// TIA Portal V16 export
// export: Created 2023-02-26T15:55:10.3538181Z, ExportSetting WithDefaults, DisplayName Totally Integrated Automation Portal, DisplayVersion V16 Update 3, DisplayName TIA Portal Version Control Interface, DisplayVersion V16 Update 2, DisplayName TIA Portal Openness, DisplayVersion V16 Update 3, DisplayName STEP 7 Professional, DisplayVersion V16 Update 3, DisplayName STEP 7 Safety, DisplayVersion V16, DisplayName WinCC Professional, DisplayVersion V16 Update 3
FUNCTION "FC19511_StdDebugInst1Order" : Void   // FC19511, LAD
TITLE = Standard Module [DEBUG] — First Order Response Simulation
{ S7_Optimized_Access := 'TRUE' }
AUTHOR : M_Gledhill
FAMILY : Debug
NAME : StdDebugInst1Order
VERSION : 0.1
// PRACTICAL SERIES AUTOMATION LIBRARY (PAL)   —   COPYRIGHT 2020 – M. GLEDHILL (MIT LICENCE)
//                   ———— ◆ ————
// FULL ONLINE DOCUMENTATION IS AVAILABLE AT: https://practicalseries.com/2001-pal/index.html
// stored: AutoNumber false, IsIECCheckEnabled true, SetENOAutomatically false, UDAEnableTagReadback false
   VAR_INPUT
      SYS_SIGNALS : "UT21000_Dy_SysSignals";   // Common system signals — logic and timing signals
      TRIGGER : Bool;   // Starts the simulation (rising edge starts the sim)
      INPUT : Real;   // The input function, x in the calculations
   END_VAR
   VAR_OUTPUT
      OUTPUT : Real;   // The output response, y in the calculations
   END_VAR
   VAR_IN_OUT
      DYNAMIC_DATA : "UT39511_Dy_DebugInst1Order";   // Dynamic data storage (UDT)
   END_VAR
   VAR_TEMP
      revInfo : "UT01000_St_SysRevision";   // Revision information for this block
      licInfo : "UT01001_St_SysLicence";   // Licensing information for this block
      act_CPUTime : DTL;   // Current CPU time (this block call)
      cal_01 : Real;   // Partial calculation see § 3.5 for details
      cal_02 : Real;   // Partial calculation see § 3.5 for details
      cal_03 : Real;   // Partial calculation see § 3.5 for details
      cal_04 : Real;   // Partial calculation see § 3.5 for details
      cal_05 : Real;   // Partial calculation see § 3.5 for details
      cal_06 : Real;   // Partial calculation see § 3.5 for details
      wrkElapsedTime : LTime;   // Working storage area (current elapsed time)
      wrkDeltaTime : LTime;   // Working storage area (current ΔT)
      wrkInt : Int;   // Working storage area (integer)
      wrkLInt : ULInt;   // Working storage area (long integer)
      wrkReal : Real;   // Working storage (real)
   END_VAR
   VAR CONSTANT
      k_NEG_MAX : Real := 3.4E-38;   // Largest negative number available to the REAL type
   END_VAR
   VAR_TEMP   // added for the SCL form of the ladder/FBD networks
      _w1 : Bool;
   END_VAR
BEGIN

REGION Network 1: Block description — Sections 1 to 2 inclusive
   // ▄▄▄▄▄▄▄▄▄▄▄▄▄▄▄▄▄▄▄▄▄▄▄▄▄▄▄▄▄▄▄▄▄  ＳＴＡＮＤＡＲＤ  ▄▄ 
   // 
   // 
   // TITLE:    DEBUG — FIRST ORDER RESPONSE SIMULATION
   // 
   // 
   // ▀▀▀▀▀▀▀▀▀▀▀▀▀▀▀▀▀▀▀▀▀▀▀▀▀▀▀▀▀▀▀▀▀▀▀▀▀▀▀▀▀▀▀▀ 
   // 
   // ┌──────────────────────────────────────────┐
   // │                                          │
   // │          FC19511 — SOFTWARE MODULE DESIGN SPECIFICATION (SMDS)            │
   // │                                          │
   // │      The PDF version of the SMDS for this module is available online here:        │
   // │              https://psop.uk/pal-smds-fc19511-p               │
   // │                                          │
   // │      It is also available as part of the Project User Defined Documentation,      │
   // │      it can be accessed by selecting this module in the Project Tree          │
   // │      (on the left) and pressing SHIFT+F1                        │
   // │                                          │
   // └─────────────────────────────────────── ʷᴵᴰ⁻ᶜᵇᶻ ┘
   // 
   // FC19511_StdDebugInst1Order is a debug simulation subroutine.
   // 
   // The module simulates a first order process reaction in response to an input signal.
   // 
   // The simulation is adjustable in terms of the system gain and the system time constant.
   // The output of the first order response simulation is in the form of a real number and is 
   // constrained to the resolution and range limits applicable to this number type within the Siemens 
   // Simatic S7-1500 controller.
   // 
   // The module will simulate a 1st order response to any type of input signal (step, ramp, sinusoid, 
   // freeform &c.).
   // 
   // The module also has a manual mode that can simulate an output at any specific time in 
   // response to a step input.
   // 
   // 
   // 
   // 
   // 
   // ▄▄▄▄▄▄▄▄▄▄▄▄▄▄▄▄▄▄▄▄▄▄▄▄▄▄▄▄▄▄▄▄▄▄▄▄▄▄▄▄▄▄▄▄
   // 1.     BLOCK TECHNICAL SUMMARY
   // 
   // 
   //  ――――――――――――――――――――――――――――――――――――――――――
   //  NOMENCLATURE & ADDRESSING
   //  ――――――――――――――――――――――――――――――――――――――――――
   //  BLOCK TITLE         1st Order Response Simulation
   //  BLOCK FUNCTION GROUP    Debug  
   //  BLOCK ADDRESS       FC19511
   //  BLOCK SYMBOL        FC19511_StdDebugInst1Order
   //  BLOCK USER ID         StdDebugInst1Order
   // 
   //  ――――――――――――――――――――――――――――――――――――――――――
   //  BLOCK TYPE & USAGE
   //  ――――――――――――――――――――――――――――――――――――――――――
   //  BLOCK TYPE         Function (FC)
   //  BLOCK NUMBER        19511
   //  LANGUAGE           LAD
   //  OPTIMISED ACCESS     Yes
   //  PAL USAGE TYPE       Standard block
   // 
   //  ――――――――――――――――――――――――――――――――――――――――――
   //  METRICS
   //  ――――――――――――――――――――――――――――――――――――――――――
   //  EXECUTION TIME        091.0 μs¹    (Note: = 14.4µs if TRIGGER is FALSE)
   //  LOAD MEMORY       46.0 kB
   //  WORK MEMORY           0.9 kB  
   //  ――――――――――――――――――――――――――――――――――――――――――
   //                ¹ Measured on: CPU-1515-2PN (order no. 6ES7512-2AM02-0AB0) 
   //                             https://psop.uk/pal-ds-cpu1515
   // 
   // 
   // 
   // ▂▂▂▂▂▂▂▂▂▂▂▂▂▂▂▂▂▂▂▂▂▂▂▂▂▂▂▂▂▂▂▂▂▂▂▂▂▂▂▂▂▂▂▂
   // 1.1      Additional referenced documents
   // 
   // 
   // In addition to the documents referenced in OB1 (section DOCUMENT REFERENCES), the 
   // following documents are associated with this module:
   // 
   // 
   //  ――――――――――――――――――――――――――――――――――――――――――
   //  REF.     DOCUMENT NO.         TITLE
   //  ――――――――――――――――――――――――――――――――――――――――――
   //  101  PS2001-5-2331-fc19511      FC19511 Calculation Sheet
   //  102  PS2001-5-2331-fc19511-011    FC19511 1st Order Response Simulation Spreadsheet
   //  ――――――――――――――――――――――――――――――――――――――――――
   // 
   // 
   // 
   //                ━━━   ⬙⬙⬙⬙⬙⬙   ━━━
   // 
   // 
   // 
   // ▄▄▄▄▄▄▄▄▄▄▄▄▄▄▄▄▄▄▄▄▄▄▄▄▄▄▄▄▄▄▄▄▄▄▄▄▄▄▄▄▄▄▄▄
   // 2.     FUNCTIONAL DESCRIPTION
   // 
   // 
   // ████████████████████████████████████████████
   // █                                          █
   // █ Note:   The following descriptions are taken from the associated Software Module     █
   // █     Design Specification [PS2001-5-2312-fc19511], the SMDS contains various     █
   // █     graphs that cannot be easily reproduced in these module comments. Where    █
   // █     essential, some rudimentary images have been included; however,        █
   // █     these are better viewed directly in the SMDS.                   █
   // █                                          █
   // █     Where images of the graphs are included, these are generated using           █
   // █     the Unicode braille characters and were generated by the following web site:     █
   // █     https://505e06b2.github.io/Image-to-Braille/                  █
   // █     (the images are 100 braille characters wide)                   █
   // █                                          █
   // █     The SMDS can be accessed directly by selecting this module (FC19511) in the     █
   // █     Project Tree (on the left) and pressing SHIFT+F1.                 █
   // █                                          █
   // █      The PDF version of the SMDS for this module is available online here:        █
   // █              https://psop.uk/pal-smds-fc19511-p               █
   // █                                          █
   // ████████████████████████████████████████████
   // 
   // FC19511 is the 1st Order Response Simulation module. The purpose of this module is to simulate 
   // a “first order” process reaction in response to an input signal.
   // 
   // First order systems are the most common type of system response for process control systems 
   // (for example the response generated when heating a tank of liquid). First order systems are often 
   // referred to as “first order lag” systems and generally reflect systems whereby the response of the 
   // system (the temperature of the water in the above example) follows the input (the temperature 
   // of the heating element) but with some delay (or lag). First order systems do not produce an 
   // oscillatory response to a step change of input and do not overshoot the input.
   // 
   // First order systems are so called because the equation linking the input to the out-put is always 
   // defined by a first order differential equation.
   // 
   // The following graphs show typical first order responses to a step change input:
   // 
   // 
   // 
   // Output y(t)
   // │⠄⠄⠄⠄⠄⠄⠄⠄⠄⠄⠄⠄⠄⠄⠄⠄⠄⠄⠄⠄⠄⠄⠄⠄⠄⠄⠄⠄⠄⠄⠄⠄⠄⠄⠄⠄⠄⠄⠄⠄⠄⠄⠄⠄⠄⠄⠄⠄⠄⠄⠄⠄⠄⠄⠄⠄⠄⠄⠄⠄⠄⠄⠄⠄⠄⠄⠄⠄⠄⠄⠄⠄⠄⠄⠄⠄⠄⠄⠄⠄⠄⠄⠄⠄⠄⠄⠄⠄⠄⠄⠄⠄⠄⠄⠄⠄⠄⠄⠄⠄
   // │⠤⠤⠤⠤⠤⠤⠤⠤⠤⠤⠤⠤⠤⠤⠤⠤⠤⠤⠤⠤⠤⠤⠤⠤⠤⠤⠤⠤⠤⠤⠤⠤⠤⠤⠤⠤⠤⠤⠤⠤⠤⠤⠤⠤⠤⠤⠤⠤⠤⠤⠤⢀⣀⣀⣀⣀⣀⣠⣤⣤⣤⣤⣤⣤⣤⣤⣤⣤⣤⣤⣤⣤⣤⣤⣤⠤⠤⠤⠤⠤⠤⠤⠤⠤⠤⠤⠤⠤⠤⠤⠤⠤⠤⠤⠤⠤⠤⠤⠤⠤
   // │⡇⠄⠄⠄⠄⠄⠄⠄⠄⠄⠄⠄⠄⠄⠄⠄⠄⠄⠄⠄⠄⠄⠄⠄⠄⠄⠄⠄⠄⠄⠄⠄⠄⠄⠄⠄⠄⠄⠄⣀⣀⣤⣤⡶⠶⠶⠒⠒⠛⠉⠉⠉⠉⠉⠉⠉⠉⠉⠉⠁⠄⠄⠄⠄⠄⠄⠄⠄⠄⠄⠄⠄⠄⠄⠄⠄⠄⠄⠄⠄⠄⠄⠄⠄⠄⠄⠄⠄⠄⠄⠄⠄⠄⠄⠄⠄⠄⠄⠄⠄
   // │⡇←— STEP INPUT  ⠄⠄⠄⠄⠄⠄⠄⠄⠄⠄⠄⠄⠄⠄⠄⠄⠄⠄⠄⠄⣀⣤⡶⠖⠚⠉⠉⠉⠁⠄⠄⠄⠄⠄⠄⠄⠄⠄⠄⠄⠄⠄⠄⠄⠄⠄⠄⠄⠄⠄⠄⠄⠄⠄⠄⠄⠄⠄⠄⠄⠄⠄⠄⠄⠄⠄⠄⠄⠄⠄⠄⠄⠄⠄⠄⠄⠄⠄⠄⠄⠄⠄⠄⠄⠄⠄⠄
   // │⡇⠄⠄⠄⠄⠄⠄⠄⠄⠄⠄⠄⠄⠄⠄⠄⠄⠄⠄⠄⠄⠄⠄⠄⠄⠄⠄⠄⢀⣠⡴⠖⠋⠉⠁⠄⠄⠄⠄⠄⠄⠄⠄⠄⠄⠄⠄⠄⠄⠄⠄⠄⠄⠄⠄⠄⠄⠄⠄⠄⠄⠄⠄⠄⠄⠄⠄⠄⠄⠄⠄⠄⠄⠄⠄⠄⠄⠄⠄⠄⠄⠄⠄⠄⠄⠄⠄⠄⠄⠄⠄⠄⠄⠄⠄⠄⠄⠄⠄⠄
   // │⡇⠄⠄⠄⠄⠄⠄⠄⠄⠄⠄⠄⠄⠄⠄⠄⠄⠄⠄⠄⠄⠄⠄⠄⠄⠄⣠⠾⠋⠄⠄⠄⠄⠄⠄⠄⠄⠄⠄⠄⠄⠄⠄⠄⠄⠄⠄⠄⠄⠄⠄⠄⠄⠄⠄⠄⠄⠄⠄⠄⠄⠄⠄⠄⠄⠄⠄⠄⠄⠄⠄⠄⠄⠄⠄⠄⠄⠄⠄⠄⠄⠄⠄⠄⠄⠄⠄⠄⠄⠄⠄⠄⠄⠄⠄⠄⠄⠄⠄⠄
   // │⡇⠄⠄⠄⠄⠄⠄⠄⠄⠄⠄⠄⠄⠄⠄⠄⠄⠄⠄⠄⠄⠄⠄⣀⡴⠋⠁⠄⠄⠄⠄⠄⠄⠄⠄⠄⠄⠄⠄⠄⠄⠄⠄⠄⠄⠄⠄⠄⠄⠄⠄⠄⠄⠄⠄⠄⠄⠄⠄⠄⠄⠄⠄⠄⠄⠄⠄⠄⠄⠄⠄⠄⠄⠄⠄⠄⠄⠄⠄⠄⠄⠄⠄⠄⠄⠄⠄⠄⠄⠄⠄⠄⠄⠄⠄⠄⠄⠄⠄⠄
   // │⡇⠄⠄⠄⠄⠄⠄⠄⠄⠄⠄⠄⠄⠄⠄⠄⠄⠄⠄⠄⠄⣠⠾⠁←— DELAYED OUTPUT  ⠄⠄⠄⠄⠄⠄⠄⠄⠄⠄⠄⠄⠄⠄⠄⠄⠄⠄⠄⠄⠄⠄⠄⠄⠄⠄⠄⠄⠄⠄⠄⠄⠄⠄⠄⠄⠄⠄⠄⠄⠄⠄⠄⠄⠄⠄⠄⠄⠄⠄⠄⠄⠄⠄⠄⠄⠄⠄
   // │⡇⠄⠄⠄⠄⠄⠄⠄⠄⠄⠄⠄⠄⠄⠄⠄⠄⠄⠄⢀⡴⠏⠄⠄⠄⠄⠄⠄⠄⠄⠄⠄⠄⠄⠄⠄⠄⠄⠄⠄⠄⠄⠄⠄⠄⠄⠄⠄⠄⠄⠄⠄⠄⠄⠄⠄⠄⠄⠄⠄⠄⠄⠄⠄⠄⠄⠄⠄⠄⠄⠄⠄⠄⠄⠄⠄⠄⠄⠄⠄⠄⠄⠄⠄⠄⠄⠄⠄⠄⠄⠄⠄⠄⠄⠄⠄⠄⠄⠄⠄
   // │⡇⠄⠄⠄⠄⠄⠄⠄⠄⠄⠄⠄⠄⠄⠄⠄⠄⢀⣴⠏⠄⠄⠄⠄⠄⠄⠄⠄⠄⠄⠄⠄⠄⠄⠄⠄⠄⠄⠄⠄⠄⠄⠄⠄⠄⠄⠄⠄⠄⠄⠄⠄⠄⠄⠄⠄⠄⠄⠄⠄⠄⠄⠄⠄⠄⠄⠄⠄⠄⠄⠄⠄⠄⠄⠄⠄⠄⠄⠄⠄⠄⠄⠄⠄⠄⠄⠄⠄⠄⠄⠄⠄⠄⠄⠄⠄⠄⠄⠄⠄
   // │⡇⠄⠄⠄⠄⠄⠄⠄⠄⠄⠄⠄⠄⠄⠄⠄⢠⡜⠃⠄⠄⠄⠄⠄⠄⠄⠄⠄⠄⠄⠄⠄⠄⠄⠄⠄⠄⠄⠄⠄⠄⠄⠄⠄⠄⠄⠄⠄⠄⠄⠄⠄⠄⠄⠄⠄⠄⠄⠄⠄⠄⠄⠄⠄⠄⠄⠄⠄⠄⠄⠄⠄⠄⠄⠄⠄⠄⠄⠄⠄⠄⠄⠄⠄⠄⠄⠄⠄⠄⠄⠄⠄⠄⠄⠄⠄⠄⠄⠄⠄
   // │⡇⠄⠄⠄⠄⠄⠄⠄⠄⠄⠄⠄⠄⠄⠄⢰⠟⠁⠄⠄⠄⠄⠄⠄⠄⠄⠄⠄⠄⠄⠄⠄⠄⠄⠄⠄⠄⠄⠄⠄⠄⠄⠄⠄⠄⠄⠄⠄⠄⠄⠄⠄⠄⠄⠄⠄⠄⠄⠄⠄⠄⠄⠄⠄⠄⠄⠄⠄⠄⠄⠄⠄⠄⠄⠄⠄⠄⠄⠄⠄⠄⠄⠄⠄⠄⠄⠄⠄⠄⠄⠄⠄⠄⠄⠄⠄⠄⠄⠄⠄
   // │⡇⠄⠄⠄⠄⠄⠄⠄⠄⠄⠄⠄⠄⠄⣰⡏⠄⠄⠄⠄⠄⠄⠄⠄⠄⠄⠄⠄⠄⠄⠄⠄⠄⠄⠄⠄⠄⠄⠄⠄⠄⠄⠄⠄⠄⠄⠄⠄⠄⠄⠄⠄⠄⠄⠄⠄⠄⠄⠄⠄⠄⠄⠄⠄⠄⠄⠄⠄⠄⠄⠄⠄⠄⠄⠄⠄⠄⠄⠄⠄⠄⠄⠄⠄⠄⠄⠄⠄⠄⠄⠄⠄⠄⠄⠄⠄⠄⠄⠄⠄
   // │⡇⠄⠄⠄⠄⠄⠄⠄⠄⠄⠄⠄⠄⢠⠏⠄⠄⠄⠄⠄⠄⠄⠄⠄⠄⠄⠄⠄⠄⠄⠄⠄⠄⠄⠄⠄⠄⠄⠄⠄⠄⠄⠄⠄⠄⠄⠄⠄⠄⠄⠄⠄⠄⠄⠄⠄⠄⠄⠄⠄⠄⠄⠄⠄⠄⠄⠄⠄⠄⠄⠄⠄⠄⠄⠄⠄⠄⠄⠄⠄⠄⠄⠄⠄⠄⠄⠄⠄⠄⠄⠄⠄⠄⠄⠄⠄⠄⠄⠄⠄
   // │⡇⠄⠄⠄⠄⠄⠄⠄⠄⠄⠄⠄⣰⡟⠄⠄⠄⠄⠄⠄⠄⠄⠄⠄⠄⠄⠄⠄⠄⠄⠄⠄⠄⠄⠄⠄⠄⠄⠄⠄⠄⠄⠄⠄⠄⠄⠄⠄⠄⠄⠄⠄⠄⠄⠄⠄⠄⠄⠄⠄⠄⠄⠄⠄⠄⠄⠄⠄⠄⠄⠄⠄⠄⠄⠄⠄⠄⠄⠄⠄⠄⠄⠄⠄⠄⠄⠄⠄⠄⠄⠄⠄⠄⠄⠄⠄⠄⠄⠄⠄
   // │⡇⠄⠄⠄⠄⠄⠄⠄⠄⠄⠄⢠⠏⠄⠄⠄⠄⠄⠄⠄⠄⠄⠄⠄⠄⠄⠄⠄⠄⠄⠄⠄⠄⠄⠄⠄⠄⠄⠄⠄⠄⠄⠄⠄⠄⠄⠄⠄⠄⠄⠄⠄⠄⠄⠄⠄⠄⠄⠄⠄⠄⠄⠄⠄⠄⠄⠄⠄⠄⠄⠄⠄⠄⠄⠄⠄⠄⠄⠄⠄⠄⠄⠄⠄⠄⠄⠄⠄⠄⠄⠄⠄⠄⠄⠄⠄⠄⠄⠄⠄
   // │⡇⠄⠄⠄⠄⠄⠄⠄⠄⠄⢠⡿⠄⠄⠄⠄⠄⠄⠄⠄⠄⠄⠄⠄⠄⠄⠄⠄⠄⠄⠄⠄⠄⠄⠄⠄⠄⠄⠄⠄⠄⠄⠄⠄⠄⠄⠄⠄⠄⠄⠄⠄⠄⠄⠄⠄⠄⠄⠄⠄⠄⠄⠄⠄⠄⠄⠄⠄⠄⠄⠄⠄⠄⠄⠄⠄⠄⠄⠄⠄⠄⠄⠄⠄⠄⠄⠄⠄⠄⠄⠄⠄⠄⠄⠄⠄⠄⠄⠄⠄
   // │⡇⠄⠄⠄⠄⠄⠄⠄⠄⠄⡿⠁⠄⠄⠄⠄⠄⠄⠄⠄⠄⠄⠄⠄⠄⠄⠄⠄⠄⠄⠄⠄⠄⠄⠄⠄⠄⠄⠄⠄⠄⠄⠄⠄⠄⠄⠄⠄⠄⠄⠄⠄⠄⠄⠄⠄⠄⠄⠄⠄⠄⠄⠄⠄⠄⠄⠄⠄⠄⠄⠄⠄⠄⠄⠄⠄⠄⠄⠄⠄⠄⠄⠄⠄⠄⠄⠄⠄⠄⠄⠄⠄⠄⠄⠄⠄⠄⠄⠄⠄
   // │⡇⠄⠄⠄⠄⠄⠄⠄⠄⣼⠃⠄⠄⠄⠄⠄⠄⠄⠄⠄⠄⠄⠄⠄⠄⠄⠄⠄⠄⠄⠄⠄⠄⠄⠄⠄⠄⠄⠄⠄⠄⠄⠄⠄⠄⠄⠄⠄⠄⠄⠄⠄⠄⠄⠄⠄⠄⠄⠄⠄⠄⠄⠄⠄⠄⠄⠄⠄⠄⠄⠄⠄⠄⠄⠄⠄⠄⠄⠄⠄⠄⠄⠄⠄⠄⠄⠄⠄⠄⠄⠄⠄⠄⠄⠄⠄⠄⠄⠄⠄
   // │⡇⠄⠄⠄⠄⠄⠄⠄⢰⡟⠄⠄⠄⠄⠄⠄⠄⠄⠄⠄⠄⠄⠄⠄⠄⠄⠄⠄⠄⠄⠄⠄⠄⠄⠄⠄⠄⠄⠄⠄⠄⠄⠄⠄⠄⠄⠄⠄⠄⠄⠄⠄⠄⠄⠄⠄⠄⠄⠄⠄⠄⠄⠄⠄⠄⠄⠄⠄⠄⠄⠄⠄⠄⠄⠄⠄⠄⠄⠄⠄⠄⠄⠄⠄⠄⠄⠄⠄⠄⠄⠄⠄⠄⠄⠄⠄⠄⠄⠄⠄
   // │⡇⠄⠄⠄⠄⠄⠄⠄⡞⠄⠄⠄⠄⠄⠄⠄⠄⠄⠄⠄⠄⠄⠄⠄⠄⠄⠄⠄⠄⠄⠄⠄⠄⠄⠄⠄⠄⠄⠄⠄⠄⠄⠄⠄⠄⠄⠄⠄⠄⠄⠄⠄⠄⠄⠄⠄⠄⠄⠄⠄⠄⠄⠄⠄⠄⠄⠄⠄⠄⠄⠄⠄⠄⠄⠄⠄⠄⠄⠄⠄⠄⠄⠄⠄⠄⠄⠄⠄⠄⠄⠄⠄⠄⠄⠄⠄⠄⠄⠄⠄
   // │⡇⠄⠄⠄⠄⠄⠄⣰⡇⠄⠄⠄⠄⠄⠄⠄⠄⠄⠄⠄⠄⠄⠄⠄⠄⠄⠄⠄⠄⠄⠄⠄⠄⠄⠄⠄⠄⠄⠄⠄⠄⠄⠄⠄⠄⠄⠄⠄⠄⠄⠄⠄⠄⠄⠄⠄⠄⠄⠄⠄⠄⠄⠄⠄⠄⠄⠄⠄⠄⠄⠄⠄⠄⠄⠄⠄⠄⠄⠄⠄⠄⠄⠄⠄⠄⠄⠄⠄⠄⠄⠄⠄⠄⠄⠄⠄⠄⠄⠄⠄
   // │⡇⠄⠄⠄⠄⠄⢰⡟⠄⠄⠄⠄⠄⠄⠄⠄⠄⠄⠄⠄⠄⠄⠄⠄⠄⠄⠄⠄⠄⠄⠄⠄⠄⠄⠄⠄⠄⠄⠄⠄⠄⠄⠄⠄⠄⠄⠄⠄⠄⠄⠄⠄⠄⠄⠄⠄⠄⠄⠄⠄⠄⠄⠄⠄⠄⠄⠄⠄⠄⠄⠄⠄⠄⠄⠄⠄⠄⠄⠄⠄⠄⠄⠄⠄⠄⠄⠄⠄⠄⠄⠄⠄⠄⠄⠄⠄⠄⠄⠄⠄
   // │⡇⠄⠄⠄⠄⠄⣸⠁⠄⠄⠄⠄⠄⠄⠄⠄⠄⠄⠄⠄⠄⠄⠄⠄⠄⠄⠄⠄⠄⠄⠄⠄⠄⠄⠄⠄⠄⠄⠄⠄⠄⠄⠄⠄⠄⠄⠄⠄⠄⠄⠄⠄⠄⠄⠄⠄⠄⠄⠄⠄⠄⠄⠄⠄⠄⠄⠄⠄⠄⠄⠄⠄⠄⠄⠄⠄⠄⠄⠄⠄⠄⠄⠄⠄⠄⠄⠄⠄⠄⠄⠄⠄⠄⠄⠄⠄⠄⠄⠄⠄
   // │⡇⠄⠄⠄⠄⢠⡇⠄⠄⠄⠄⠄⠄⠄⠄⠄⠄⠄⠄⠄⠄⠄⠄⠄⠄⠄⠄⠄⠄⠄⠄⠄⠄⠄⠄⠄⠄⠄⠄⠄⠄⠄⠄⠄⠄⠄⠄⠄⠄⠄⠄⠄⠄⠄⠄⠄⠄⠄⠄⠄⠄⠄⠄⠄⠄⠄⠄⠄⠄⠄⠄⠄⠄⠄⠄⠄⠄⠄⠄⠄⠄⠄⠄⠄⠄⠄⠄⠄⠄⠄⠄⠄⠄⠄⠄⠄⠄⠄⠄⠄
   // │⡇⠄⠄⠄⠄⣿⠃⠄⠄⠄⠄⠄⠄⠄⠄⠄⠄⠄⠄⠄⠄⠄⠄⠄⠄⠄⠄⠄⠄⠄⠄⠄⠄⠄⠄⠄⠄⠄⠄⠄⠄⠄⠄⠄⠄⠄⠄⠄⠄⠄⠄⠄⠄⠄⠄⠄⠄⠄⠄⠄⠄⠄⠄⠄⠄⠄⠄⠄⠄⠄⠄⠄⠄⠄⠄⠄⠄⠄⠄⠄⠄⠄⠄⠄⠄⠄⠄⠄⠄⠄⠄⠄⠄⠄⠄⠄⠄⠄⠄⠄
   // │⡇⠄⠄⠄⢸⡏⠄⠄⠄⠄⠄⠄⠄⠄⠄⠄⠄⠄⠄⠄⠄⠄⠄⠄⠄⠄⠄⠄⠄⠄⠄⠄⠄⠄⠄⠄⠄⠄⠄⠄⠄⠄⠄⠄⠄⠄⠄⠄⠄⠄⠄⠄⠄⠄⠄⠄⠄⠄⠄⠄⠄⠄⠄⠄⠄⠄⠄⠄⠄⠄⠄⠄⠄⠄⠄⠄⠄⠄⠄⠄⠄⠄⠄⠄⠄⠄⠄⠄⠄⠄⠄⠄⠄⠄⠄⠄⠄⠄⠄⠄
   // │⡇⠄⠄⠄⣸⠁⠄⠄⠄⠄⠄⠄⠄⠄⠄⠄⠄⠄⠄⠄⠄⠄⠄⠄⠄⠄⠄⠄⠄⠄⠄⠄⠄⠄⠄⠄⠄⠄⠄⠄⠄⠄⠄⠄⠄⠄⠄⠄⠄⠄⠄⠄⠄⠄⠄⠄⠄⠄⠄⠄⠄⠄⠄⠄⠄⠄⠄⠄⠄⠄⠄⠄⠄⠄⠄⠄⠄⠄⠄⠄⠄⠄⠄⠄⠄⠄⠄⠄⠄⠄⠄⠄⠄⠄⠄⠄⠄⠄⠄⠄
   // │⡇⠄⠄⢠⡇⠄⠄⠄⠄⠄⠄⠄⠄⠄⠄⠄⠄⠄⠄⠄⠄⠄⠄⠄⠄⠄⠄⠄⠄⠄⠄⠄⠄⠄⠄⠄⠄⠄⠄⠄⠄⠄⠄⠄⠄⠄⠄⠄⠄⠄⠄⠄⠄⠄⠄⠄⠄⠄⠄⠄⠄⠄⠄⠄⠄⠄⠄⠄⠄⠄⠄⠄⠄⠄⠄⠄⠄⠄⠄⠄⠄⠄⠄⠄⠄⠄⠄⠄⠄⠄⠄⠄⠄⠄⠄⠄⠄⠄⠄⠄
   // │⡇⠄⠄⣼⠇⠄⠄⠄⠄⠄⠄⠄⠄⠄⠄⠄⠄⠄⠄⠄⠄⠄⠄⠄⠄⠄⠄⠄⠄⠄⠄⠄⠄⠄⠄⠄⠄⠄⠄⠄⠄⠄⠄⠄⠄⠄⠄⠄⠄⠄⠄⠄⠄⠄⠄⠄⠄⠄⠄⠄⠄⠄⠄⠄⠄⠄⠄⠄⠄⠄⠄⠄⠄⠄⠄⠄⠄⠄⠄⠄⠄⠄⠄⠄⠄⠄⠄⠄⠄⠄⠄⠄⠄⠄⠄⠄⠄⠄⠄⠄
   // │⡇⠄⠄⡿⠄⠄⠄⠄⠄⠄⠄⠄⠄⠄⠄⠄⠄⠄⠄⠄⠄⠄⠄⠄⠄⠄⠄⠄⠄⠄⠄⠄⠄⠄⠄⠄⠄⠄⠄⠄⠄⠄⠄⠄⠄⠄⠄⠄⠄⠄⠄⠄⠄⠄⠄⠄⠄⠄⠄⠄⠄⠄⠄⠄⠄⠄⠄⠄⠄⠄⠄⠄⠄⠄⠄⠄⠄⠄⠄⠄⠄⠄⠄⠄⠄⠄⠄⠄⠄⠄⠄⠄⠄⠄⠄⠄⠄⠄⠄⠄
   // │⡇⠄⢰⠃⠄⠄⠄⠄⠄⠄⠄⠄⠄⠄⠄⠄⠄⠄⠄⠄⠄⠄⠄⠄⠄⠄⠄⠄⠄⠄⠄⠄⠄⠄⠄⠄⠄⠄⠄⠄⠄⠄⠄⠄⠄⠄⠄⠄⠄⠄⠄⠄⠄⠄⠄⠄⠄⠄⠄⠄⠄⠄⠄⠄⠄⠄⠄⠄⠄⠄⠄⠄⠄⠄⠄⠄⠄⠄⠄⠄⠄⠄⠄⠄⠄⠄⠄⠄⠄⠄⠄⠄⠄⠄⠄⠄⠄⠄⠄⠄
   // │⡇⠄⣾⠄⠄⠄⠄⠄⠄⠄⠄⠄⠄⠄⠄⠄⠄⠄⠄⠄⠄⠄⠄⠄⠄⠄⠄⠄⠄⠄⠄⠄⠄⠄⠄⠄⠄⠄⠄⠄⠄⠄⠄⠄⠄⠄⠄⠄⠄⠄⠄⠄⠄⠄⠄⠄⠄⠄⠄⠄⠄⠄⠄⠄⠄⠄⠄⠄⠄⠄⠄⠄⠄⠄⠄⠄⠄⠄⠄⠄⠄⠄⠄⠄⠄⠄⠄⠄⠄⠄⠄⠄⠄⠄⠄⠄⠄⠄⠄⠄
   // │⡇⢰⡟⠄⠄⠄⠄⠄⠄⠄⠄⠄⠄⠄⠄⠄⠄⠄⠄⠄⠄⠄⠄⠄⠄⠄⠄⠄⠄⠄⠄⠄⠄⠄⠄⠄⠄⠄⠄⠄⠄⠄⠄⠄⠄⠄⠄⠄⠄⠄⠄⠄⠄⠄⠄⠄⠄⠄⠄⠄⠄⠄⠄⠄⠄⠄⠄⠄⠄⠄⠄⠄⠄⠄⠄⠄⠄⠄⠄⠄⠄⠄⠄⠄⠄⠄⠄⠄⠄⠄⠄⠄⠄⠄⠄⠄⠄⠄⠄⠄
   // │⡇⣾⠇⠄⠄⠄⠄⠄⠄⠄⠄⠄⠄⠄⠄⠄⠄⠄⠄⠄⠄⠄⠄⠄⠄⠄⠄⠄⠄⠄⠄⠄⠄⠄⠄⠄⠄⠄⠄⠄⠄⠄⠄⠄⠄⠄⠄⠄⠄⠄⠄⠄⠄⠄⠄⠄⠄⠄⠄⠄⠄⠄⠄⠄⠄⠄⠄⠄⠄⠄⠄⠄⠄⠄⠄⠄⠄⠄⠄⠄⠄⠄⠄⠄⠄⠄⠄⠄⠄⠄⠄⠄⠄⠄⠄⠄⠄⠄⠄⠄
   // │⡇⡿⠄⠄⠄⠄⠄⠄⠄⠄⠄⠄⠄⠄⠄⠄⠄⠄⠄⠄⠄⠄⠄⠄⠄⠄⠄⠄⠄⠄⠄⠄⠄⠄⠄⠄⠄⠄⠄⠄⠄⠄⠄⠄⠄⠄⠄⠄⠄⠄⠄⠄⠄⠄⠄⠄⠄⠄⠄⠄⠄⠄⠄⠄⠄⠄⠄⠄⠄⠄⠄⠄⠄⠄⠄⠄⠄⠄⠄⠄⠄⠄⠄⠄⠄⠄⠄⠄⠄⠄⠄⠄⠄⠄⠄⠄⠄⠄⠄⠄
   // │⡇⠃⠄⠄⠄⠄⠄⠄⠄⠄⠄⠄⠄⠄⠄⠄⠄⠄⠄⠄⠄⠄⠄⠄⠄⠄⠄⠄⠄⠄⠄⠄⠄⠄⠄⠄⠄⠄⠄⠄⠄⠄⠄⠄⠄⠄⠄⠄⠄⠄⠄⠄⠄⠄⠄⠄⠄⠄⠄⠄⠄⠄⠄⠄⠄⠄⠄⠄⠄⠄⠄⠄⠄⠄⠄⠄⠄⠄⠄⠄⠄⠄⠄⠄⠄⠄⠄⠄⠄⠄⠄⠄⠄⠄⠄⠄⠄⠄⠄⠄
   // ┼ ─ ─ ─ ─ ─ ─ ─ ─ ─ ─ ─ ─ ─ ─ ─ ─ ─ ─ ─ ─ ─ ─ ─ ─ ─ ─ ─ ─ ─ ─ ─ ─ ─ ─ ─ ─ ─ ─ ─ ─ ─ ─  ─ ─ ─ ─    Time (t)
   // 
   // 
   // 
   // ▂▂▂▂▂▂▂▂▂▂▂▂▂▂▂▂▂▂▂▂▂▂▂▂▂▂▂▂▂▂▂▂▂▂▂▂▂▂▂▂▂▂▂▂
   // 2.1      Scope and limitations of the simulation
   // 
   // 
   // The first order response simulation will provide a real time response for a first order simulation.
   // 
   // The simulation will be adjustable in terms of the system gain (K) and the time constant of the 
   // system (τ).
   // 
   // The output of the first order response simulation will be in the form of a real number.
   // 
   // 
   // 
   // 
   // ▁▁▁▁▁▁▁▁▁▁▁▁▁▁▁▁▁▁▁▁▁▁▁▁▁▁▁▁▁▁▁▁▁▁▁▁▁▁▁▁▁▁▁▁
   // 2.1.1     The limitations of the simulation
   // 
   // 
   // The output of the second order response simulation will be in the form of a real number and will 
   // be constrained to the limits applicable to this number type within the Siemens controller.
   // 
   // The S7-1500 range of Controllers supports real numbers as values, these are 32-bit numbers 
   // and, within a Controller, have the following range limits:
   // 
   // 
   //  ――――――――――――――――――――――――――――――――――――――――――
   //              LOWER RANGE LIMIT     UPPER RANGE LIMIT
   //  ――――――――――――――――――――――――――――――――――――――――――
   //  S7-1500 real number:     ±3.402323×10^(-38)           ±3.402323×10^(+38)
   //  ――――――――――――――――――――――――――――――――――――――――――
   // 
   // This range is considered acceptable for all practical uses of the module.
   // 
   // 
   // 
   // ▁▁▁▁▁▁▁▁▁▁▁▁▁▁▁▁▁▁▁▁▁▁▁▁▁▁▁▁▁▁▁▁▁▁▁▁▁▁▁▁▁▁▁▁
   // 2.1.2     The nature of the simulation calculations
   // 
   // 
   // The module will generate the correct responses for any first order system. The module uses a 
   // discrete time approximation calculation to determine the correct output for any given input. The 
   // calculation is an iterative algorithm, the formulae for which is derived in full in the associated 
   // calculations sheet [Ref. 101], available here:
   // 
   //          https://psop.uk/pal-calc-fc19511-p
   // 
   // These calculations are based around the mathematical functions available to the Controller 
   // (these are in addition to the standard mathematical operations: addition, subtraction, 
   // multiplication and division).
   // 
   // Each Controller supports the following common mathematical functions:
   // 
   // 
   //  ――――――――――――――――――――――――――――――――――――――――――
   //  OPERATION    EXAMPLE         DESCRIPTION
   //  ――――――――――――――――――――――――――――――――――――――――――
   //  SQR        x^2          Form the square
   //  SQRT         √x            Form the square root
   //  EXP        e^x          Exponential
   //  LN          log_e(⁡x)        Natural logarithm
   //  SIN         sin(⁡x)         Sine
   //  ASIN          sin^-1(x)          Arcsine, inverse sine
   //  COS          cos(⁡x)        Cosine
   //  ACOS        cos^-1(x)         Arccosine, inverse cosine
   //  TAN           tan(⁡x)         Tangent
   //  ATAN         tan^-1(x)         Arctangent, inverse tangent
   //  ABS        |x|            Modulus
   //  ――――――――――――――――――――――――――――――――――――――――――
   //  Table 2.1 S7 Controller — common mathematical functions
   // 
   // 
   // 
   // ▂▂▂▂▂▂▂▂▂▂▂▂▂▂▂▂▂▂▂▂▂▂▂▂▂▂▂▂▂▂▂▂▂▂▂▂▂▂▂▂▂▂▂▂
   // 2.2      The second order response
   // 
   // 
   // The response of a second order system (y) to an input (x) is defined using the general form of a 
   // second order system transfer function, this is expressed below in the time domain as a second 
   // order differential equation (see the calculation sheet [Ref. 101], Appendix B for details):
   // 
   //                 dy
   //             τ ----- ┼  y  =  Kx  (2.1)
   //                 dt
   // 
   // Where:    K is the system gain
   //      τ is referred to as the system time constant (seconds)
   // 
   // 
   // 
   // ▂▂▂▂▂▂▂▂▂▂▂▂▂▂▂▂▂▂▂▂▂▂▂▂▂▂▂▂▂▂▂▂▂▂▂▂▂▂▂▂▂▂▂▂
   // 2.3      The calculations
   // 
   // 
   // Two forms of calculation are needed to produce a model for a first order system. The first being a 
   // continuous simulation running in real-time with a varying or constant input signal.
   // 
   // The second being the discrete result for a step input under manual conditions (i.e. a fixed input 
   // and specific time are provided and a single, corresponding output value generated).
   // 
   // Both of these calculations are discussed in the following sections:
   // 
   // 
   // 
   // ▁▁▁▁▁▁▁▁▁▁▁▁▁▁▁▁▁▁▁▁▁▁▁▁▁▁▁▁▁▁▁▁▁▁▁▁▁▁▁▁▁▁▁▁
   // 2.3.1     Real-time simulation calculation for any input type
   // 
   // 
   // The normal operation of the module (in automatic mode) is to produce a continuous real-time 
   // model of a first order system that once triggered, runs continuously, producing an output 
   // response that mimics a first order system responding to a variable (or constant) input as time 
   // progresses, the simulation continues until the triggering condition is removed.
   // 
   // The calculation needed to produce a first order system response to any type of input signal is 
   // best achieved using a discrete time approximation method. The details of this method are given 
   // in [Ref. 101], Section 2.1, and the results are given below:
   // 
   // The final form of the calculations that will be used in the FC19511 software module for a real time 
   // simulation to any input type is:
   // 
   //    y[n] = Ka x[n]  ┼ (1-a) y[n-1]  (2.2)
   // 
   //              ΔT
   //    where:   a = ----------
   //            τ+ΔT
   // 
   //    K is the system gain (a constant number)
   //    τ is the system time constant (in seconds)
   //    Δt is the sampling interval between calculations (in seconds)
   //    x[n] is the input at the current iteration 
   //    y[n] is the output at the current iteration 
   //    y[n-1] is the output at the previous iteration 
   // 
   // 
   // It should be noted that this is an iterative algorithm, the previous value of the output must 
   // be retained between calculations.
   // 
   // For best results, Δt should be very much smaller than the system time constant, i.e.:
   // 
   //                    τ
   //    Δt ≪ τ      Typically, Δt ≤ ----
   //                      10
   // 
   // Note also, that Δt need not be constant between samples.
   // 
   // 
   // 
   // ▁▁▁▁▁▁▁▁▁▁▁▁▁▁▁▁▁▁▁▁▁▁▁▁▁▁▁▁▁▁▁▁▁▁▁▁▁▁▁▁▁▁▁▁
   // 2.3.2     Manual simulation calculation for a step input at a particular time
   // 
   // 
   // In manual mode, an instantaneous calculation is carried out using the first order equation at a 
   // particular time and for a particular input value.
   // 
   // Since, under manual control, both the time and the input are fixed single values, it is not possible 
   // to determine the nature of the input (i.e. is it a ramp, sinusoid &c.), hence for all manual 
   // operations within the simulation, the input is considered to be a step input that changed to the 
   // manually specified input value at time = 0, and that prior to this the input was zero¹. I.e. a step 
   // input that changed from zero to the specified value at time = 0.
   // 
   // To produce a specific output value in response to a fixed step input at a particular time, it is 
   // necessary to solve the first order differential equation given in equation (2.1), as a non-iterative, 
   // discreate calculation. To do this, it is necessary to convert the equation into the Laplace domain² 
   // (using standard Laplace transforms, see [Ref. 101], Appendix A) algebraically solve the equation 
   // and then convert the result back to the time domain (using the standard inverse Laplace 
   // transforms, again see [Ref. 101], Appendix A).
   // 
   // The final form of the manual calculations that will be used in the FC19511 software module for a 
   // single point input type is:
   // 
   //          ┌      -t/τ  ┐
   //    y(t) = KX│ 1 ─  e   │
   //          └       ┘
   // 
   //    K is the system gain (a constant number)
   //    τ is the system time constant (in seconds)
   //    X is the fixed input value
   // 
   // 
   // ――――――――――
   // ¹         A step response is the most common type of response
   // 
   // ²         The calculation sheet associated with this module [Ref. 101], explains the Laplace 
   //      transform mechanisms and how they are used within the calculations necessary for 
   //      the functioning of this module. Further explanation of the Laplace transform is not 
   //      given in this document, again the reader is referred to the calculation 
   //      sheet [Ref. 101].
   // ――――――――――
   // 
   // 
   // 
   // ▁▁▁▁▁▁▁▁▁▁▁▁▁▁▁▁▁▁▁▁▁▁▁▁▁▁▁▁▁▁▁▁▁▁▁▁▁▁▁▁▁▁▁▁
   // 2.3.3     Calculation spreadsheet model
   // 
   // 
   // An accompanying spreadsheet [Ref. 016] is available, this allows all the various responses to be 
   // graphically simulated with adjustable values (it was this spreadsheet that produced the various 
   // response plots used within this document), this spreadsheet is available here:
   // 
   //      http://psop.uk/pal-calc-fc19511-p
   // 
   // 
   // 
   // ▂▂▂▂▂▂▂▂▂▂▂▂▂▂▂▂▂▂▂▂▂▂▂▂▂▂▂▂▂▂▂▂▂▂▂▂▂▂▂▂▂▂▂▂
   // 2.4      Real-time responses for typical inputs
   // 
   // 
   // First order systems respond to various types of input (step, ramp, sinusoidal) in very predictable 
   // ways. First order systems never produce oscillatory responses (unless the input itself is 
   // oscillating) and never overshoot the input (cf. 2nd order systems, see FC19512). The general 
   // response of a first order system is that of an inherent delay (or lag) in the response of the output 
   // compared with the input.
   // 
   // This inherent delay is reflected in the system time constant (τ), measured in seconds.
   // 
   // The following sections consider how the system time constant affects the output for several 
   // typical input types:
   // 
   // 
   // STEP INPUT
   // 
   // │⠄⠄⠄⠄⠄⠄⠄⠄⠄⠄⠄⠄⠄⠄⠄⠄⠄⠄⠄⠄⠄⠄⠄τ = 20s⠄⠄⠄⠄⠄⠄⠄⠄⠄⠄⠄⠄⠄⠄⠄⠄⠄⠄⠄⠄⠄⠄⠄⠄⠄⠄⠄⠄⠄⠄⠄⠄⠄⠄⠄⠄⠄⠄⠄⠄⠄⠄⠄⠄⠄⠄⠄⠄⠄⠄⠄⠄⠄⠄⠄⠄⠄⠄⠄⠄⠄⠄⠄⠄⠄⠄⠄⠄⠄⠄⠄⠄
   // X─ ─ ─ ─ ─ ─ ─ ─ ─ ─ ─ ─ ─ ─ ─ ─ ─ ─ ─ ─ ─ ─ ─ ─ ─ ─ ─ ─ ─ ─ ─ ─ ─ ─ ─ ─ ─ ─ ─ ─ ─ ─ ─ ─ ─ ─ ─
   // │⠄⠄⠄⠄⠄⠄⠄⠄⠄⠄⠄⠄⠄⠄⠄⠄⠄⠄⠄⠄⠄⠄⠄⠄⠄⠄⠄⠄⠄⠄⠄⠄⠄⠄⠄⠄⠄⠄⠄⠄⠄⠄⠄⠄⠄⠄⠄⠄⠄⠄⠄⠄⠄⠄⠄⠄⠄⠄⠄⠄⠄⣀⣀⣀⣀⣠⣤⡤⠤⠤⠶⠶⠶⠶⠒⠒⠒⠒⠚⠛⠛⠛⠛⠉⠉⠉⠉⠉⠉⠉⠉⠉⠉⠉⠉⠉⠉⠉⠉⠉
   // │⠄⠄⠄⠄⠄⠄⠄⠄⠄⠄⠄⠄⠄⠄⠄⠄⠄⠄⠄⠄⠄⠄⠄⠄⠄⠄⠄⠄⠄⠄⠄⠄⠄⠄⠄⠄⠄⠄⠄⠄⠄⠄⠄⠄⠄⠄⠄⠄⠄⠄⢀⣀⣠⡤⠤⠶⠖⠒⠛⠄⠄⠄⠄⠄⠄⠄⠄⠄⠄⠄⠄⠄⠄⠄99% of steady state ─ ─ ─ ─ ╎⠄
   // │⠄⠄⠄⠄⠄⠄⠄⠄⠄⠄⠄⠄⠄⠄⠄⠄⠄⠄⠄⠄⠄⠄⠄⠄⠄⠄⠄⠄⠄⠄⠄⠄⠄⠄⠄⠄⠄⠄⠄⠄⠄⠄⠄⢀⣀⣠⠴⠖⠚⠋⠉⠁⠄⠄⠄⠄⠄⠄⠄⠄⠄⠄⠄⠄⠄⠄⠄⠄⠄⠄⠄⠄⠄⠄⠄⠄⠄⠄⠄⠄⠄⠄⠄⠄⠄⠄⠄⠄⠄⠄⠄⠄⠄⠄⠄⠄⠄⠄╎⠄
   // │⠄⠄⠄⠄⠄⠄⠄⠄⠄⠄⠄⠄⠄⠄⠄⠄⠄⠄⠄⠄⠄⠄⠄⠄⠄⠄⠄⠄⠄⠄⠄⠄⠄⠄⠄⠄⠄⠄⢀⣠⡤⠖⠚⠉⠁⠄⠄⠄⠄⠄⠄⠄⠄⠄⠄⠄⠄⠄⠄⠄⠄⠄⠄⠄⠄⠄⠄⠄⠄⠄⠄⠄⠄⠄⠄⠄⠄⠄⠄⠄⠄⠄⠄⠄⠄⠄⠄⠄⠄⠄⠄⠄⠄⠄⠄⠄⠄⠄╎⠄
   // │⠄⠄⠄⠄⠄⠄⠄⠄⠄⠄⠄⠄⠄⠄⠄⠄⠄⠄⠄⠄⠄⠄⠄⠄⠄⠄⠄⠄⠄⠄⠄⠄⠄⠄⠄⣠⡴⠚⠋⠁⠄⠄⠄⠄⠄⠄⠄⠄⠄⠄⠄⠄⠄⠄⠄⠄⠄⠄⠄⠄⠄⠄⠄⠄⠄⠄⠄⠄⠄⠄⠄⠄⠄⠄⠄⠄⠄⠄⠄⠄⠄⠄⠄⠄⠄⠄⠄⠄⠄⠄⠄⠄⠄⠄⠄⠄⠄⠄╎⠄
   // │⠄⠄⠄⠄⠄⠄⠄⠄⠄⠄⠄⠄⠄⠄⠄⠄⠄⠄⠄⠄⠄⠄⠄⠄⠄⠄⠄⠄⠄⠄⠄⢀⣠⠖⠋⠁⠄⠄⠄⠄⠄⠄⠄⠄⠄⠄⠄⠄⠄⠄⠄⠄⠄⠄⠄⠄⠄⠄⠄⠄⠄⠄⠄⠄⠄⠄⠄⠄⠄⠄⠄⠄⠄⠄⠄⠄⠄⠄⠄⠄⠄⠄⠄⠄⠄⠄⠄⠄⠄⠄⠄⠄⠄⠄⠄⠄⠄⠄╎⠄
   // │⠄⠄⠄⠄⠄⠄⠄⠄⠄⠄⠄⠄⠄⠄⠄⠄⠄⠄⠄⠄⠄⠄⠄⠄⠄⠄⠄⠄⠄⣠⠴⠋⠄⠄⠄⠄⠄⠄⠄⠄⠄⠄⠄⠄⠄⠄⠄⠄⠄⠄⠄⠄⠄⠄⠄⠄⠄⠄⠄⠄⠄⠄⠄⠄⠄⠄⠄⠄⠄⠄⠄⠄⠄⠄⠄⠄⠄⠄⠄⠄⠄⠄⠄⠄⠄⠄⠄⠄⠄⠄⠄⠄⠄⠄⠄⠄⠄⠄╎⠄
   // │⠄⠄⠄⠄⠄⠄⠄⠄⠄⠄⠄⠄⠄⠄⠄⠄⠄⠄⠄⠄⠄⠄⠄⠄⠄⠄⢀⡤⠚⠁⠄⠄⠄⠄⠄⠄⠄⠄⠄⠄⠄⠄⠄⠄⠄⠄⠄⠄⠄⠄⠄⠄⠄⠄⠄⠄⠄⠄⠄⠄⠄⠄⠄⠄⠄⠄⠄⠄⠄⠄⠄⠄⠄⠄⠄⠄⠄⠄⠄⠄⠄⠄⠄⠄⠄⠄⠄⠄⠄⠄⠄⠄⠄⠄⠄⠄⠄⠄╎⠄
   // │⠄⠄⠄⠄⠄⠄⠄⠄⠄⠄⠄⠄⠄⠄⠄⠄⠄⠄⠄⠄⠄⠄⠄⠄⢀⡴⠋⠄⠄⠄⠄⠄⠄⠄⠄⠄⠄⠄⠄⠄⠄⠄⠄⠄⠄⠄⠄⠄⠄⠄⠄⠄⠄⠄⠄⠄⠄⠄⠄⠄⠄⠄⠄⠄⠄⠄⠄⠄⠄⠄⠄⠄⠄⠄⠄⠄⠄⠄⠄⠄⠄⠄⠄⠄⠄⠄⠄⠄⠄⠄⠄⠄⠄⠄⠄⠄⠄⠄╎⠄
   // │⠄⠄⠄⠄⠄⠄⠄⠄⠄⠄⠄⠄⠄⠄⠄⠄⠄⠄⠄⠄⠄⠄⢀⡴⠋⠄⠄⠄⠄⠄⠄⠄⠄⠄⠄⠄⠄⠄⠄⠄⠄⠄⠄⠄⠄⠄⠄⠄⠄⠄⠄⠄⠄⠄⠄⠄⠄⠄⠄⠄⠄⠄⠄⠄⠄⠄⠄⠄⠄⠄⠄⠄⠄⠄⠄⠄⠄⠄⠄⠄⠄⠄⠄⠄⠄⠄⠄⠄⠄⠄⠄⠄⠄⠄⠄⠄⠄⠄╎⠄
   // │⠄⠄⠄⠄⠄⠄⠄⠄⠄⠄⠄⠄⠄⠄⠄⠄⠄⠄⠄⠄⠄⣠⠋⠄⠄⠄⠄⠄⠄⠄⠄⠄⠄⠄⠄⠄⠄⠄⠄⠄⠄⠄⠄⠄⠄⠄⠄⠄⠄⠄⠄⠄⠄⠄⠄⠄⠄⠄⠄⠄⠄⠄⠄⠄⠄⠄⠄⠄⠄⠄⠄⠄⠄⠄⠄⠄⠄⠄⠄⠄⠄⠄⠄⠄⠄⠄⠄⠄⠄⠄⠄⠄⠄⠄⠄⠄⠄⠄╎⠄
   // │⠄⠄⠄⠄⠄⠄⠄⠄⠄⠄⠄⠄⠄⠄⠄⠄⠄⠄⠄⢀⠞⠁⠄⠄⠄⠄⠄⠄⠄⠄⠄⠄⠄⠄⠄⠄⠄⠄⠄⠄⠄⠄⠄⠄⠄⠄⠄⠄⠄⠄⠄⠄⠄⠄⠄⠄⠄⠄⠄⠄⠄⠄⠄⠄⠄⠄⠄⠄⠄⠄⠄⠄⠄⠄⠄⠄⠄⠄⠄⠄⠄⠄⠄⠄⠄⠄⠄⠄⠄⠄⠄⠄⠄⠄⠄⠄⠄⠄╎⠄
   // │⠄⠄⠄⠄⠄⠄⠄⠄⠄⠄⠄⠄⠄⠄⠄⠄⠄⠄⣴⠋─ ─ ─ ─ ─  63% of steady state  ⠄⠄⠄⠄⠄⠄⠄⠄⠄⠄⠄⠄⠄⠄⠄⠄⠄⠄⠄⠄⠄⠄⠄⠄⠄⠄⠄⠄⠄⠄⠄⠄⠄⠄⠄⠄⠄⠄⠄⠄⠄⠄⠄⠄⠄⠄⠄⠄⠄⠄⠄╎⠄
   // │⠄⠄⠄⠄⠄⠄⠄⠄⠄⠄⠄⠄⠄⠄⠄⠄⢀⡾⠁⠄⠄⠄⠄⠄⠄⠄⠄⠄⠄⠄⠄⠄⠄⠄⠄⠄⠄⠄⠄⠄⠄⠄⠄⠄⠄⠄⠄⠄⠄⠄⠄⠄⠄⠄⠄⠄⠄⠄⠄⠄⠄⠄⠄⠄⠄⠄⠄⠄⠄⠄⠄⠄⠄⠄⠄⠄⠄⠄⠄⠄⠄⠄⠄⠄⠄⠄⠄⠄⠄⠄⠄⠄⠄⠄⠄⠄⠄⠄╎⠄
   // │⠄⠄⠄⠄⠄⠄⠄⠄⠄⠄⠄⠄⠄⠄⠄⢠⠞⠄ ╎⠄⠄⠄⠄⠄⠄⠄⠄⠄⠄⠄⠄⠄⠄⠄⠄⠄⠄⠄⠄⠄⠄⠄⠄⠄⠄⠄⠄⠄⠄⠄⠄⠄⠄⠄⠄⠄⠄⠄⠄⠄⠄⠄⠄⠄⠄⠄⠄⠄⠄⠄⠄⠄⠄⠄⠄⠄⠄⠄⠄⠄⠄⠄⠄⠄⠄⠄⠄⠄⠄⠄⠄⠄⠄⠄⠄⠄⠄╎⠄
   // │⠄⠄⠄⠄⠄⠄⠄⠄⠄⠄⠄⠄⠄⠄⣠⠏⠄⠄ ╎⠄⠄⠄⠄⠄⠄⠄⠄⠄⠄⠄⠄⠄⠄⠄⠄⠄⠄⠄⠄⠄⠄⠄⠄⠄⠄⠄⠄⠄⠄⠄⠄⠄⠄⠄⠄⠄⠄⠄⠄⠄⠄⠄⠄⠄⠄⠄⠄⠄⠄⠄⠄⠄⠄⠄⠄⠄⠄⠄⠄⠄⠄⠄⠄⠄⠄⠄⠄⠄⠄⠄⠄⠄⠄⠄⠄⠄⠄╎⠄
   // │⠄⠄⠄⠄⠄⠄⠄⠄⠄⠄⠄⠄⠄⣰⠋⠄⠄⠄ ╎⠄⠄⠄⠄⠄⠄⠄⠄⠄⠄⠄⠄⠄⠄⠄⠄⠄⠄⠄⠄⠄⠄⠄⠄⠄⠄⠄⠄⠄⠄⠄⠄⠄⠄⠄⠄⠄⠄⠄⠄⠄⠄⠄⠄⠄⠄⠄⠄⠄⠄⠄⠄⠄⠄⠄⠄⠄⠄⠄⠄⠄⠄⠄⠄⠄⠄⠄⠄⠄⠄⠄⠄⠄⠄⠄⠄⠄⠄╎⠄
   // │⠄⠄⠄⠄⠄⠄⠄⠄⠄⠄⠄⠄⣰⠃⠄⠄⠄⠄ ╎⠄⠄⠄⠄⠄⠄⠄⠄⠄⠄⠄⠄⠄⠄⠄⠄⠄⠄⠄⠄⠄⠄⠄⠄⠄⠄⠄⠄⠄⠄⠄⠄⠄⠄⠄⠄⠄⠄⠄⠄⠄⠄⠄⠄⠄⠄⠄⠄⠄⠄⠄⠄⠄⠄⠄⠄⠄⠄⠄⠄⠄⠄⠄⠄⠄⠄⠄⠄⠄⠄⠄⠄⠄⠄⠄⠄⠄⠄╎⠄
   // │⠄⠄⠄⠄⠄⠄⠄⠄⠄⠄⠄⣸⠃⠄⠄⠄⠄⠄ ╎⠄⠄⠄⠄⠄⠄⠄⠄⠄⠄⠄⠄⠄⠄⠄⠄⠄⠄⠄⠄⠄⠄⠄⠄⠄⠄⠄⠄⠄⠄⠄⠄⠄⠄⠄⠄⠄⠄⠄⠄⠄⠄⠄⠄⠄⠄⠄⠄⠄⠄⠄⠄⠄⠄⠄⠄⠄⠄⠄⠄⠄⠄⠄⠄⠄⠄⠄⠄⠄⠄⠄⠄⠄⠄⠄⠄⠄⠄╎⠄
   // │⠄⠄⠄⠄⠄⠄⠄⠄⠄⠄⣰⠃⠄⠄⠄⠄⠄⠄ ╎⠄⠄⠄⠄⠄⠄⠄⠄⠄⠄⠄⠄⠄⠄⠄⠄⠄⠄⠄⠄⠄⠄⠄⠄⠄⠄⠄⠄⠄⠄⠄⠄⠄⠄⠄⠄⠄⠄⠄⠄⠄⠄⠄⠄⠄⠄⠄⠄⠄⠄⠄⠄⠄⠄⠄⠄⠄⠄⠄⠄⠄⠄⠄⠄⠄⠄⠄⠄⠄⠄⠄⠄⠄⠄⠄⠄⠄⠄╎⠄
   // │⠄⠄⠄⠄⠄⠄⠄⠄⠄⣰⠃⠄⠄⠄⠄⠄⠄⠄ ╎⠄⠄⠄⠄⠄⠄⠄⠄⠄⠄⠄⠄⠄⠄⠄⠄⠄⠄⠄⠄⠄⠄⠄⠄⠄⠄⠄⠄⠄⠄⠄⠄⠄⠄⠄⠄⠄⠄⠄⠄⠄⠄⠄⠄⠄⠄⠄⠄⠄⠄⠄⠄⠄⠄⠄⠄⠄⠄⠄⠄⠄⠄⠄⠄⠄⠄⠄⠄⠄⠄⠄⠄⠄⠄⠄⠄⠄⠄╎⠄
   // │⠄⠄⠄⠄⠄⠄⠄⠄⢰⠇⠄⠄⠄⠄⠄⠄⠄⠄ ╎⠄⠄⠄⠄⠄⠄⠄⠄⠄⠄⠄⠄⠄⠄⠄⠄⠄⠄⠄⠄⠄⠄⠄⠄⠄⠄⠄⠄⠄⠄⠄⠄⠄⠄⠄⠄⠄⠄⠄⠄⠄⠄⠄⠄⠄⠄⠄⠄⠄⠄⠄⠄⠄⠄⠄⠄⠄⠄⠄⠄⠄⠄⠄⠄⠄⠄⠄⠄⠄⠄⠄⠄⠄⠄⠄⠄⠄⠄╎⠄
   // │⠄⠄⠄⠄⠄⠄⠄⢠⡏⠄⠄⠄⠄⠄⠄⠄⠄⠄ ╎⠄⠄⠄⠄⠄⠄⠄⠄⠄⠄⠄⠄⠄⠄⠄⠄⠄⠄⠄⠄⠄⠄⠄⠄⠄⠄⠄⠄⠄⠄⠄⠄⠄⠄⠄⠄⠄⠄⠄⠄⠄⠄⠄⠄⠄⠄⠄⠄⠄⠄⠄⠄⠄⠄⠄⠄⠄⠄⠄⠄⠄⠄⠄⠄⠄⠄⠄⠄⠄⠄⠄⠄⠄⠄⠄⠄⠄⠄╎⠄
   // │⠄⠄⠄⠄⠄⠄⠄⡞⠄⠄⠄⠄⠄⠄⠄⠄⠄⠄ ╎⠄⠄⠄⠄⠄⠄⠄⠄⠄⠄⠄⠄⠄⠄⠄⠄⠄⠄⠄⠄⠄⠄⠄⠄⠄⠄⠄⠄⠄⠄⠄⠄⠄⠄⠄⠄⠄⠄⠄⠄⠄⠄⠄⠄⠄⠄⠄⠄⠄⠄⠄⠄⠄⠄⠄⠄⠄⠄⠄⠄⠄⠄⠄⠄⠄⠄⠄⠄⠄⠄⠄⠄⠄⠄⠄⠄⠄⠄╎⠄
   // │⠄⠄⠄⠄⠄⠄⣸⠃⠄⠄⠄⠄⠄⠄⠄⠄⠄⠄ ╎⠄⠄⠄⠄⠄⠄⠄⠄⠄⠄⠄⠄⠄⠄⠄⠄⠄⠄⠄⠄⠄⠄⠄⠄⠄⠄⠄⠄⠄⠄⠄⠄⠄⠄⠄⠄⠄⠄⠄⠄⠄⠄⠄⠄⠄⠄⠄⠄⠄⠄⠄⠄⠄⠄⠄⠄⠄⠄⠄⠄⠄⠄⠄⠄⠄⠄⠄⠄⠄⠄⠄⠄⠄⠄⠄⠄⠄⠄╎⠄
   // │⠄⠄⠄⠄⠄⢰⠇⠄⠄⠄⠄⠄⠄⠄⠄⠄⠄⠄ ╎⠄⠄⠄⠄⠄⠄⠄⠄⠄⠄⠄⠄⠄⠄⠄⠄⠄⠄⠄⠄⠄⠄⠄⠄⠄⠄⠄⠄⠄⠄⠄⠄⠄⠄⠄⠄⠄⠄⠄⠄⠄⠄⠄⠄⠄⠄⠄⠄⠄⠄⠄⠄⠄⠄⠄⠄⠄⠄⠄⠄⠄⠄⠄⠄⠄⠄⠄⠄⠄⠄⠄⠄⠄⠄⠄⠄⠄⠄╎⠄
   // │⠄⠄⠄⠄⢀⡟⠄⠄⠄⠄⠄⠄⠄⠄⠄⠄⠄⠄ ╎⠄⠄⠄⠄⠄⠄⠄⠄⠄⠄⠄⠄⠄⠄⠄⠄⠄⠄⠄⠄⠄⠄⠄⠄⠄⠄⠄⠄⠄⠄⠄⠄⠄⠄⠄⠄⠄⠄⠄⠄⠄⠄⠄⠄⠄⠄⠄⠄⠄⠄⠄⠄⠄⠄⠄⠄⠄⠄⠄⠄⠄⠄⠄⠄⠄⠄⠄⠄⠄⠄⠄⠄⠄⠄⠄⠄⠄⠄╎⠄
   // │⠄⠄⠄⠄⡼⠁⠄⠄⠄⠄⠄⠄⠄⠄⠄⠄⠄⠄ ╎⠄⠄⠄⠄⠄⠄⠄⠄⠄⠄⠄⠄⠄⠄⠄⠄⠄⠄⠄⠄⠄⠄⠄⠄⠄⠄⠄⠄⠄⠄⠄⠄⠄⠄⠄⠄⠄⠄⠄⠄⠄⠄⠄⠄⠄⠄⠄⠄⠄⠄⠄⠄⠄⠄⠄⠄⠄⠄⠄⠄⠄⠄⠄⠄⠄⠄⠄⠄⠄⠄⠄⠄⠄⠄⠄⠄⠄⠄╎⠄
   // │⠄⠄⠄⢰⠇⠄⠄⠄⠄⠄⠄⠄⠄⠄⠄⠄⠄⠄ ╎⠄⠄⠄⠄⠄⠄⠄⠄⠄⠄⠄⠄⠄⠄⠄⠄⠄⠄⠄⠄⠄⠄⠄⠄⠄⠄⠄⠄⠄⠄⠄⠄⠄⠄⠄⠄⠄⠄⠄⠄⠄⠄⠄⠄⠄⠄⠄⠄⠄⠄⠄⠄⠄⠄⠄⠄⠄⠄⠄⠄⠄⠄⠄⠄⠄⠄⠄⠄⠄⠄⠄⠄⠄⠄⠄⠄⠄⠄╎⠄
   // │⠄⠄⢀⡏⠄⠄⠄⠄⠄⠄⠄⠄⠄⠄⠄⠄⠄⠄ ╎⠄⠄⠄⠄⠄⠄⠄⠄⠄⠄⠄⠄⠄⠄⠄⠄⠄⠄⠄⠄⠄⠄⠄⠄⠄⠄⠄⠄⠄⠄⠄⠄⠄⠄⠄⠄⠄⠄⠄⠄⠄⠄⠄⠄⠄⠄⠄⠄⠄⠄⠄⠄⠄⠄⠄⠄⠄⠄⠄⠄⠄⠄⠄⠄⠄⠄⠄⠄⠄⠄⠄⠄⠄⠄⠄⠄⠄⠄╎⠄
   // │⠄⠄⡼⠁⠄⠄⠄⠄⠄⠄⠄⠄⠄⠄⠄⠄⠄⠄ ╎⠄⠄⠄⠄⠄⠄⠄⠄⠄⠄⠄⠄⠄⠄⠄⠄⠄⠄⠄⠄⠄⠄⠄⠄⠄⠄⠄⠄⠄⠄⠄⠄⠄⠄⠄⠄⠄⠄⠄⠄⠄⠄⠄⠄⠄⠄⠄⠄⠄⠄⠄⠄⠄⠄⠄⠄⠄⠄⠄⠄⠄⠄⠄⠄⠄⠄⠄⠄⠄⠄⠄⠄⠄⠄⠄⠄⠄⠄╎⠄
   // │⠄⣸⠃⠄⠄⠄⠄⠄⠄⠄⠄⠄⠄⠄⠄⠄⠄⠄ ╎⠄⠄⠄⠄⠄⠄⠄⠄⠄⠄⠄⠄⠄⠄⠄⠄⠄⠄⠄⠄⠄⠄⠄⠄⠄⠄⠄⠄⠄⠄⠄⠄⠄⠄⠄⠄⠄⠄⠄⠄⠄⠄⠄⠄⠄⠄⠄⠄⠄⠄⠄⠄⠄⠄⠄⠄⠄⠄⠄⠄⠄⠄⠄⠄⠄⠄⠄⠄⠄⠄⠄⠄⠄⠄⠄⠄⠄⠄╎⠄
   // │⡴⠃⠄⠄⠄⠄⠄⠄⠄⠄⠄⠄⠄⠄⠄⠄⠄⠄ ╎⠄⠄⠄⠄⠄⠄⠄⠄⠄⠄⠄⠄⠄⠄⠄⠄⠄⠄⠄⠄⠄⠄⠄⠄⠄⠄⠄⠄⠄⠄⠄⠄⠄⠄⠄⠄⠄⠄⠄⠄⠄⠄⠄⠄⠄⠄⠄⠄⠄⠄⠄⠄⠄⠄⠄⠄⠄⠄⠄⠄⠄⠄⠄⠄⠄⠄⠄⠄⠄⠄⠄⠄⠄⠄⠄⠄⠄⠄╎⠄
   // ┼ ─ ─ ─ ─ ┼ ─ ─ ─ ─ ┼ ─ ─ ─ ─ ┼ ─ ─ ─ ─ ┼ ─ ─ ─ ─ ┼ ─ ─ ─ ─ ┼ ─ ─ ─ ─ ┼ ─ ─ ─ ─ ┼ ─ ─ ─ ─ ┼ ─ ─ ─ ─ ┼
   // 0.0     10       20       30       40       50       60       70       80       90      100 s
   //               τ                                               5τ
   //    Increasing τ gives a slower response.
   // 
   //                1
   //    Initial rate of change = ---   Time to reach 63% of input (X) = τ   Time to reach steady state = 5τ
   //                τ
   // 
   // 
   // RAMP INPUT
   // 
   // │⠄⠄⠄⠄⠄⠄⠄⠄⠄⠄⠄⠄⠄⠄⠄⠄⠄⠄⠄⠄⠄⠄⠄τ = 20s ⠄⠄⠄⠄⠄⠄⠄⠄⠄⠄⠄⠄⠄⠄⠄⠄⠄⠄⠄⠄⠄⠄⠄⠄⠄⠄⠄⠄⠄⠄⠄⠄⠄⠄⠄⠄⠄⠄⠄⠄⠄⠄⠄⠄⠄⠄⠄⠄⠄⠄⠄⠄⠄⠄⠄⠄⠄⠄⠄⠄⠄⠄⠄⠄⠄⠄⠄⠄⢀⡠⠔
   // │⠄⠄⠄⠄⠄⠄⠄⠄⠄⠄⠄⠄⠄⠄⠄⠄⠄⠄⠄⠄⠄⠄⠄⠄⠄⠄⠄⠄⠄⠄⠄⠄⠄⠄⠄⠄⠄⠄⠄⠄⠄⠄⠄⠄⠄⠄⠄⠄⠄⠄⠄⠄⠄⠄⠄⠄⠄⠄⠄⠄⠄⠄⠄⠄⠄⠄⠄⠄⠄⠄⠄⠄⠄⠄⠄⠄⠄⠄⠄⠄⠄⠄⠄⠄⠄⠄⠄⠄⠄⠄⠄⠄⠄⢀⣠⠴⠊⠉⠄⠄
   // │⠄⠄⠄⠄⠄⠄⠄⠄⠄⠄⠄⠄⠄⠄⠄⠄⠄⠄⠄⠄⠄⠄⠄⠄⠄⠄⠄⠄⠄⠄⠄⠄⠄⠄⠄⠄⠄⠄⠄⠄⠄⠄⠄⠄⠄⠄⠄⠄⠄⠄⠄⠄⠄⠄⠄⠄⠄⠄⠄⠄⠄⠄⠄⠄⠄⠄⠄⠄⠄⠄⠄⠄⠄⠄⠄⠄⠄⠄⠄⠄⠄⠄⠄⠄⠄⠄⠄⠄⠄⢀⣀⠴⠊⠉⠄⠄⠄⠄⠄⠄
   // │⠄⠄⠄⠄⠄⠄⠄⠄⠄⠄⠄⠄⠄⠄⠄⠄⠄⠄⠄⠄⠄⠄⠄⠄⠄⠄⠄⠄⠄⠄⠄⠄⠄⠄⠄⠄⠄⠄⠄⠄⠄⠄⠄⠄⠄⠄⠄⠄⠄⠄⠄⠄⠄⠄⠄⠄⠄⠄⠄⠄⠄⠄⠄⠄⠄⠄⠄⠄⠄⠄⠄⠄⠄⠄⠄⠄⠄⠄⠄⠄⠄⠄⠄⠄⠄⠄⣀⡤⠒⠋← ─ INPUT
   // │⠄⠄⠄⠄⠄⠄⠄⠄⠄⠄⠄⠄⠄⠄⠄⠄⠄⠄⠄⠄⠄⠄⠄⠄⠄⠄⠄⠄⠄⠄⠄⠄⠄⠄⠄⠄⠄⠄⠄⠄⠄⠄⠄⠄⠄⠄⠄⠄⠄⠄⠄⠄⠄⠄⠄⠄⠄⠄⠄⠄⠄⠄⠄⠄⠄⠄⠄⠄⠄⠄⠄⠄⠄⠄⠄⠄⠄⠄⠄⠄⠄⠄⢀⡤⠖⠋⠁⠄⠄⠄⠄⠄⠄⠄⠄⠄⠄⠄⠄⠄
   // │⠄⠄⠄⠄⠄⠄⠄⠄⠄⠄⠄⠄⠄⠄⠄⠄⠄⠄⠄⠄⠄⠄⠄⠄⠄⠄⠄⠄⠄⠄⠄⠄⠄⠄⠄⠄⠄⠄⠄⠄⠄⠄⠄⠄⠄⠄⠄⠄⠄⠄⠄⠄⠄⠄⠄⠄⠄⠄⠄⠄⠄⠄⠄⠄⠄⠄⠄⠄⠄⠄⠄⠄⠄⠄⠄⠄⠄⠄⢀⣠⠔⠊⠁⠄⠄⠄⠄⠄⠄⠄⠄⠄⠄⠄⠄⠄⠄⣀⣤⡾
   // │⠄⠄⠄⠄⠄⠄⠄⠄⠄⠄⠄⠄⠄⠄⠄⠄⠄⠄⠄⠄⠄⠄⠄⠄⠄⠄⠄⠄⠄⠄⠄⠄⠄⠄⠄⠄⠄⠄⠄⠄⠄⠄⠄⠄⠄⠄⠄⠄⠄⠄⠄⠄⠄⠄⠄⠄⠄⠄⠄⠄⠄⠄⠄⠄⠄⠄⠄⠄⠄⠄⠄⠄⠄⠄⢀⣠⠔⠚⠁← ─ ─  τ  ─ ─→⢀⣤⡶⠟⠋⠄⠄
   // │⠄⠄⠄⠄⠄⠄⠄⠄⠄⠄⠄⠄⠄⠄⠄⠄⠄⠄⠄⠄⠄⠄⠄⠄⠄⠄⠄⠄⠄⠄⠄⠄⠄⠄⠄⠄⠄⠄⠄⠄⠄⠄⠄⠄⠄⠄⠄⠄⠄⠄⠄⠄⠄⠄⠄⠄⠄⠄⠄⠄⠄⠄⠄⠄⠄⠄⠄⠄⠄⠄⠄⣠⠤⠚⠉⠄⠄⠄⠄⠄⠄⠄⠄⠄⠄⠄⠄⠄⠄⢀⣤⡶⠟⠋⠁⠄⠄⠄⠄⠄
   // │⠄⠄⠄⠄⠄⠄⠄⠄⠄⠄⠄⠄⠄⠄⠄⠄⠄⠄⠄⠄⠄⠄⠄⠄⠄⠄⠄⠄⠄⠄⠄⠄⠄⠄⠄⠄⠄⠄⠄⠄⠄⠄⠄⠄⠄⠄⠄⠄⠄⠄⠄⠄⠄⠄⠄⠄⠄⠄⠄⠄⠄⠄⠄⠄⠄⠄⠄⣀⡤⠒⠉⠄⠄⠄⠄⠄⠄⠄⠄⠄⠄⠄⠄⠄⠄⢀⣠⣴⠞⠋⠁⠄⠄⠄⠄⠄⠄⠄⠄⠄
   // │⠄⠄⠄⠄⠄⠄⠄⠄⠄⠄⠄⠄⠄⠄⠄⠄⠄⠄⠄⠄⠄⠄⠄⠄⠄⠄⠄⠄⠄⠄⠄⠄⠄⠄⠄⠄⠄⠄⠄⠄⠄⠄⠄⠄⠄⠄⠄⠄⠄⠄⠄⠄⠄⠄⠄⠄⠄⠄⠄⠄⠄⠄⠄⣀⡤⠖⠋⠄⠄⠄⠄⠄⠄⠄⠄⠄⠄⠄⠄⠄⠄⢀⣠⣴⠞⠛⠁← ─ OUTPUT
   // │⠄⠄⠄⠄⠄⠄⠄⠄⠄⠄⠄⠄⠄⠄⠄⠄⠄⠄⠄⠄⠄⠄⠄⠄⠄⠄⠄⠄⠄⠄⠄⠄⠄⠄⠄⠄⠄⠄⠄⠄⠄⠄⠄⠄⠄⠄⠄⠄⠄⠄⠄⠄⠄⠄⠄⠄⠄⠄⠄⣀⡠⠴⠊⠁⠄⠄⠄⠄⠄⠄⠄⠄⠄⠄⠄⠄⠄⢀⣀⣤⠶⠛⠉⠄⠄⠄⠄⠄⠄⠄⠄⠄⠄⠄⠄⠄⠄⠄⠄⠄
   // │⠄⠄⠄⠄⠄⠄⠄⠄⠄⠄⠄⠄⠄⠄⠄⠄⠄⠄⠄⠄⠄⠄⠄⠄⠄⠄⠄⠄⠄⠄⠄⠄⠄⠄⠄⠄⠄⠄⠄⠄⠄⠄⠄⠄⠄⠄⠄⠄⠄⠄⠄⠄⠄⠄⠄⢀⣀⠴⠊⠁⠄⠄⠄⠄⠄⠄⠄⠄⠄⠄⠄⠄⠄⠄⣀⣴⠶⠛⠉⠄⠄⠄⠄⠄⠄⠄⠄⠄⠄⠄⠄⠄⠄⠄⠄⠄⠄⠄⠄⠄
   // │⠄⠄⠄⠄⠄⠄⠄⠄⠄⠄⠄⠄⠄⠄⠄⠄⠄⠄⠄⠄⠄⠄⠄⠄⠄⠄⠄⠄⠄⠄⠄⠄⠄⠄⠄⠄⠄⠄⠄⠄⠄⠄⠄⠄⠄⠄⠄⠄⠄⠄⠄⠄⣀⠴⠚⠉⠄⠄⠄⠄⠄⠄⠄⠄⠄⠄⠄⠄⠄⠄⣀⣴⠶⠛⠉⠄⠄⠄⠄⠄⠄⠄⠄⠄⠄⠄⠄⠄⠄⠄⠄⠄⠄⠄⠄⠄⠄⠄⠄⠄
   // │⠄⠄⠄⠄⠄⠄⠄⠄⠄⠄⠄⠄⠄⠄⠄⠄⠄⠄⠄⠄⠄⠄⠄⠄⠄⠄⠄⠄⠄⠄⠄⠄⠄⠄⠄⠄⠄⠄⠄⠄⠄⠄⠄⠄⠄⠄⠄⠄⣀⡤⠒⠉⠁⠄⠄⠄⠄⠄⠄⠄⠄⠄⠄⠄⠄⠄⣀⣤⠶⠟⠉⠁⠄⠄⠄⠄⠄⠄⠄⠄⠄⠄⠄⠄⠄⠄⠄⠄⠄⠄⠄⠄⠄⠄⠄⠄⠄⠄⠄⠄
   // │⠄⠄⠄⠄⠄⠄⠄⠄⠄⠄⠄⠄⠄⠄⠄⠄⠄⠄⠄⠄⠄⠄⠄⠄⠄⠄⠄⠄⠄⠄⠄⠄⠄⠄⠄⠄⠄⠄⠄⠄⠄⠄⠄⠄⣀⡤⠖⠋⠁⠄⠄⠄⠄⠄⠄⠄⠄⠄⠄⠄⠄⠄⣀⣤⡶⠟⠉⠁⠄⠄⠄⠄⠄⠄⠄⠄⠄⠄⠄⠄⠄⠄⠄⠄⠄⠄⠄⠄⠄⠄⠄⠄⠄⠄⠄⠄⠄⠄⠄⠄
   // │⠄⠄⠄⠄⠄⠄⠄⠄⠄⠄⠄⠄⠄⠄⠄⠄⠄⠄⠄⠄⠄⠄⠄⠄⠄⠄⠄⠄⠄⠄⠄⠄⠄⠄⠄⠄⠄⠄⠄⠄⢀⡠⠖⠋⠁⠄⠄⠄⠄⠄⠄⠄⠄⠄⠄⠄⠄⠄⣀⣤⡶⠞⠋⠁⠄⠄⠄⠄⠄⠄⠄⠄⠄⠄⠄⠄⠄⠄⠄⠄⠄⠄⠄⠄⠄⠄⠄⠄⠄⠄⠄⠄⠄⠄⠄⠄⠄⠄⠄⠄
   // │⠄⠄⠄⠄⠄⠄⠄⠄⠄⠄⠄⠄⠄⠄⠄⠄⠄⠄⠄⠄⠄⠄⠄⠄⠄⠄⠄⠄⠄⠄⠄⠄⠄⠄⠄⠄⠄⣠⠖⠊⠉⠄⠄⠄⠄⠄⠄⠄⠄⠄⠄⠄⠄⠄⣀⣤⡶⠟⠉⠁⠄⠄⠄⠄⠄⠄⠄⠄⠄⠄⠄⠄⠄⠄⠄⠄⠄⠄⠄⠄⠄⠄⠄⠄⠄⠄⠄⠄⠄⠄⠄⠄⠄⠄⠄⠄⠄⠄⠄⠄
   // │⠄⠄⠄⠄⠄⠄⠄⠄⠄⠄⠄⠄⠄⠄⠄⠄⠄⠄⠄⠄⠄⠄⠄⠄⠄⠄⠄⠄⠄⠄⠄⠄⠄⣠⠤⠚⠉⠄⠄⠄⠄⠄⠄⠄⠄⠄⠄⠄⠄⠄⢀⣤⡶⠟⠋⠁⠄⠄⠄⠄⠄⠄⠄⠄⠄⠄⠄⠄⠄⠄⠄⠄⠄⠄⠄⠄⠄⠄⠄⠄⠄⠄⠄⠄⠄⠄⠄⠄⠄⠄⠄⠄⠄⠄⠄⠄⠄⠄⠄⠄
   // │⠄⠄⠄⠄⠄⠄⠄⠄⠄⠄⠄⠄⠄⠄⠄⠄⠄⠄⠄⠄⠄⠄⠄⠄⠄⠄⠄⠄⠄⣀⡤⠖⠋⠄⠄⠄⠄⠄⠄⠄⠄⠄⠄⠄⠄⠄⣀⣤⡶⠟⠋⠁⠄⠄⠄⠄⠄⠄⠄⠄⠄⠄⠄⠄⠄⠄⠄⠄⠄⠄⠄⠄⠄⠄⠄⠄⠄⠄⠄⠄⠄⠄⠄⠄⠄⠄⠄⠄⠄⠄⠄⠄⠄⠄⠄⠄⠄⠄⠄⠄
   // │⠄⠄⠄⠄⠄⠄⠄⠄⠄⠄⠄⠄⠄⠄⠄⠄⠄⠄⠄⠄⠄⠄⠄⠄⠄⣀⡤⠖⠋⠄⠄⠄⠄⠄⠄⠄⠄⠄⠄⠄⠄⢀⣠⣤⠾⠛⠉⠄⠄⠄⠄⠄⠄⠄⠄⠄⠄⠄⠄⠄⠄⠄⠄⠄⠄⠄⠄⠄⠄⠄⠄⠄⠄⠄⠄⠄⠄⠄⠄⠄⠄⠄⠄⠄⠄⠄⠄⠄⠄⠄⠄⠄⠄⠄⠄⠄⠄⠄⠄⠄
   // │⠄⠄⠄⠄⠄⠄⠄⠄⠄⠄⠄⠄⠄⠄⠄⠄⠄⠄⠄⠄⠄⢀⣠⠔⠋⠁⠄⠄⠄⠄⠄⠄⠄⠄⠄⠄⠄⢀⣤⡴⠞⠛⠉⠄⠄⠄⠄⠄⠄⠄⠄⠄⠄⠄⠄⠄⠄⠄⠄⠄⠄⠄⠄⠄⠄⠄⠄⠄⠄⠄⠄⠄⠄⠄⠄⠄⠄⠄⠄⠄⠄⠄⠄⠄⠄⠄⠄⠄⠄⠄⠄⠄⠄⠄⠄⠄⠄⠄⠄⠄
   // │⠄⠄⠄⠄⠄⠄⠄⠄⠄⠄⠄⠄⠄⠄⠄⠄⠄⢀⣠⠔⠋⠁⠄⠄⠄⠄⠄⠄⠄⠄⠄⠄⢀⣠⣤⡶⠟⠋⠁⠄⠄⠄⠄⠄⠄⠄⠄⠄⠄⠄⠄⠄⠄⠄⠄⠄⠄⠄⠄⠄⠄⠄⠄⠄⠄⠄⠄⠄⠄⠄⠄⠄⠄⠄⠄⠄⠄⠄⠄⠄⠄⠄⠄⠄⠄⠄⠄⠄⠄⠄⠄⠄⠄⠄⠄⠄⠄⠄⠄⠄
   // │⠄⠄⠄⠄⠄⠄⠄⠄⠄⠄⠄⠄⠄⠄⣠⠴⠚⠉⠄⠄⠄⠄⠄⠄⠄⠄⠄⠄⣀⣤⡶⠞⠛⠉⠄⠄⠄⠄⠄⠄⠄⠄⠄⠄⠄⠄⠄⠄⠄⠄⠄⠄⠄⠄⠄⠄⠄⠄⠄⠄⠄⠄⠄⠄⠄⠄⠄⠄⠄⠄⠄⠄⠄⠄⠄⠄⠄⠄⠄⠄⠄⠄⠄⠄⠄⠄⠄⠄⠄⠄⠄⠄⠄⠄⠄⠄⠄⠄⠄⠄
   // │⠄⠄⠄⠄⠄⠄⠄⠄⠄⠄⣀⠤⠖⠉⠄⠄⠄⠄⠄⠄⠄⠄⢀⣀⣤⡶⠿⠛⠉⠄⠄⠄⠄⠄⠄⠄⠄⠄⠄⠄⠄⠄⠄⠄⠄⠄⠄⠄⠄⠄⠄⠄⠄⠄⠄⠄⠄⠄⠄⠄⠄⠄⠄⠄⠄⠄⠄⠄⠄⠄⠄⠄⠄⠄⠄⠄⠄⠄⠄⠄⠄⠄⠄⠄⠄⠄⠄⠄⠄⠄⠄⠄⠄⠄⠄⠄⠄⠄⠄⠄
   // │⠄⠄⠄⠄⠄⠄⢀⡠⠖⠉⠁⠄⠄⠄⠄⠄⢀⣀⣠⣤⠶⠞⠋⠉⠁⠄⠄⠄⠄⠄⠄⠄⠄⠄⠄⠄⠄⠄⠄⠄⠄⠄⠄⠄⠄⠄⠄⠄⠄⠄⠄⠄⠄⠄⠄⠄⠄⠄⠄⠄⠄⠄⠄⠄⠄⠄⠄⠄⠄⠄⠄⠄⠄⠄⠄⠄⠄⠄⠄⠄⠄⠄⠄⠄⠄⠄⠄⠄⠄⠄⠄⠄⠄⠄⠄⠄⠄⠄⠄⠄
   // │⠄⠄⢀⡠⠖⠊⠁⠄⠄⣀⣀⣠⣤⠶⠶⠛⠋⠉⠉⠄⠄⠄⠄⠄⠄⠄⠄⠄⠄⠄⠄⠄⠄⠄⠄⠄⠄⠄⠄⠄⠄⠄⠄⠄⠄⠄⠄⠄⠄⠄⠄⠄⠄⠄⠄⠄⠄⠄⠄⠄⠄⠄⠄⠄⠄⠄⠄⠄⠄⠄⠄⠄⠄⠄⠄⠄⠄⠄⠄⠄⠄⠄⠄⠄⠄⠄⠄⠄⠄⠄⠄⠄⠄⠄⠄⠄⠄⠄⠄⠄
   // │⠴⠾⠿⠶⠶⠶⠞⠛⠛⠉⠉⠁⠄⠄⠄⠄⠄⠄⠄⠄⠄⠄⠄⠄⠄⠄⠄⠄⠄⠄⠄⠄⠄⠄⠄⠄⠄⠄⠄⠄⠄⠄⠄⠄⠄⠄⠄⠄⠄⠄⠄⠄⠄⠄⠄⠄⠄⠄⠄⠄⠄⠄⠄⠄⠄⠄⠄⠄⠄⠄⠄⠄⠄⠄⠄⠄⠄⠄⠄⠄⠄⠄⠄⠄⠄⠄⠄⠄⠄⠄⠄⠄⠄⠄⠄⠄⠄⠄⠄⠄
   // ┼ ─ ─ ─ ─ ┼ ─ ─ ─ ─ ┼ ─ ─ ─ ─ ┼ ─ ─ ─ ─ ┼ ─ ─ ─ ─ ┼ ─ ─ ─ ─ ┼ ─ ─ ─ ─ ┼ ─ ─ ─ ─ ┼ ─ ─ ─ ─ ┼ ─ ─ ─ ─ ┼
   // 0.0     10       20       30       40       50       60       70       80       90      100 s
   // 
   //    Increasing τ gives a slower response.
   // 
   //    Output follows input with a lag = τ   Time to reach steady state = 5τ
   // 
   // 
   // SINUSOIDAL INPUT
   // 
   // │⠄τ = 10s ⠄⠄⠄⠄⠄⠄⠄⠄⠄⠄⠄⠄⠄⠄⠄⠄⣀⣀⣀⣀⠄← ─ INPUT ⠄⠄⠄⠄⠄⠄⠄⠄⠄⠄⠄⠄⠄⠄⠄⠄⠄⠄⠄⠄⠄⠄⠄⠄⠄⠄⠄⠄⠄⠄⠄⠄⠄⠄⠄⠄⠄⠄⠄⠄⠄⠄⠄⠄⠄⠄⠄⠄⠄⠄⠄⠄⠄⠄⠄⠄⠄⠄⠄⠄⠄⠄⠄
   // │⠄⠄⠄⠄⠄⠄⠄⠄⠄⠄⠄⠄⠄⠄⠄⠄⠄⠄⠄⣠⠔⠚⠉⠄⠄⠄⠈⠉⠒⢤⡀⠄⠄⠄⠄⠄⠄⠄⠄⠄⠄⠄⠄⠄⠄⠄⠄⠄⠄⠄⠄⠄⠄⠄⠄⠄⠄⠄⠄⠄⠄⠄⠄⠄⠄⠄⠄⠄⠄⠄⠄⠄⠄⠄⠄⠄⠄⠄⠄⠄⠄⠄⠄⠄⠄⠄⠄⠄⠄⠄⠄⠄⠄⠄⠄⠄⠄⠄⠄⠄
   // │⠄⠄⠄⠄⠄⠄⠄⠄⠄⠄⠄⠄⠄⠄⠄⠄⠄⣠⠞⠁⠄⠄⠄⠄⠄⠄⠄⠄⠄⠄⠉⠦⡀⠄⠄⠄⠄⠄⠄⠄⠄⠄⠄⠄⠄⠄⠄⠄⠄⠄⠄⠄⠄⠄⠄⠄⠄⠄⠄⠄⠄⠄⠄⠄⠄⠄⠄⠄⠄⠄⠄⠄⠄⠄⠄⠄⠄⠄⠄⠄⠄⠄⠄⠄⠄⠄⠄⠄⠄⠄⠄⠄⠄⠄⠄⠄⠄⠄⠄⠄
   // │⠄⠄⠄⠄⠄⠄⠄⠄⠄⠄⠄⠄⠄⠄⠄⢀⠞⠁⠄⠄⠄⠄⠄⠄⠄⠄⣀⣤⠶⠛⠛⠉⠙⢟⠳⠶⣄⡀⠄⠄⠄⠄⠄⠄⠄⠄⠄⠄⠄⠄⠄⠄⠄⠄⠄⠄⠄⠄⠄⠄⠄⠄⠄⠄⠄⠄⠄⠄⠄⠄⠄⠄⠄⠄⠄⠄⠄⠄⠄⠄⠄⠄⠄⠄⠄⠄⠄⠄⠄⠄⠄⠄⠄⠄⠄⠄⠄⠄⠄⠄
   // │⠄⠄⠄⠄⠄⠄⠄⠄⠄⠄⠄⠄⠄⠄⣠⠋⠄⠄⠄⠄⠄⠄⠄⠄⣠⠾⠋⠄⠄⠄⠄⠄⠄⠄⠳⡀⠈⠙⢶⣄⠄⠄⠄⠄⠄⠄⠄⠄⠄⠄⠄⠄⠄⠄⠄⠄⠄⠄⠄⠄⠄⠄⠄⠄⠄⠄⠄⠄⠄⠄⠄⠄⠄⠄⠄⠄⠄⠄⠄⠄⠄⠄⠄⠄⠄⠄⠄⠄⠄⠄⠄⠄⠄⠄⠄⠄⠄⠄⠄⠄
   // │⠄⠄⠄⠄⠄⠄⠄⠄⠄⠄⠄⠄⢀⡔⠁⠄⠄⠄⠄⠄⠄⠄⣠⠞⠁⠄⠄⠄⠄⠄⠄⠄⠄⠄⠄⠙⣄⠄⠄⠙⢷⣄⠄← ─ OUTPUT  ⠄⠄⠄⠄⠄⠄⠄⠄⠄⠄⠄⠄⠄⠄⠄⠄⠄⠄⠄⠄⠄⠄⠄⠄⠄⠄⠄⠄⠄⠄⠄⠄⠄⠄⠄⠄⠄⠄⠄⠄⠄⠄⠄⠄⠄⠄
   // │⠄⠄⠄⠄⠄⠄⠄⠄⠄⠄⠄⢀⡞⠄⠄⠄⠄⠄⠄⠄⣠⡞⠁⠄⠄⠄⠄⠄⠄⠄⠄⠄⠄⠄⠄⠄⠘⢆⠄⠄⠄⠙⣦⡀⠄⠄⠄⠄⠄⠄⠄⠄⠄⠄⠄⠄⠄⠄⠄⠄⠄⠄⠄⠄⠄⠄⠄⠄⠄⠄⠄⠄⠄⠄⠄⠄⠄⠄⠄⠄⠄⠄⠄⠄⠄⠄⠄⠄⠄⠄⠄⠄⠄⠄⠄⠄⠄⠄⠄⠄
   // │⠄⠄⠄⠄⠄⠄⠄⠄⠄⠄⢀⠞⠄⠄⠄⠄⠄⠄⢀⣼⠋⠄⠄⠄⠄⠄⠄⠄⠄⠄⠄⠄⠄⠄⠄⠄⠄⠈⢦⠄⠄⠄⠈⢳⣄⠄⠄⠄⠄⠄⠄⠄⠄⠄⠄⠄⠄⠄⠄⠄⠄⠄⠄⠄⠄⠄⠄⠄⠄⠄⠄⠄⠄⠄⠄⠄⠄⠄⠄⠄⠄⠄⠄⠄⠄⠄⠄⠄⠄⠄⠄⠄⠄⠄⠄⠄⠄⠄⠄⠄
   // │⠄⠄⠄⠄⠄⠄⠄⠄⠄⢀⡎⠄⠄⠄⠄⠄⠄⢠⡿⠁⠄⠄⠄⠄⠄⠄⠄⠄⠄⠄⠄⠄⠄⠄⠄⠄⠄⠄⠈⢇⠄⠄⠄⠄⠻⣆⠄⠄⠄⠄⠄⠄⠄⠄⠄⠄⠄⠄⠄⠄⠄⠄⠄⠄⠄⠄⠄⠄⠄⠄⠄⠄⠄⠄⠄⠄⠄⠄⠄⠄⠄⠄⠄⠄⠄⠄⠄⠄⠄⠄⠄⠄⠄⠄⠄⠄⠄⠄⠄⠄
   // │⠄⠄⠄⠄⠄⠄⠄⠄⢀⠎⠄⠄⠄⠄⠄⠄⣴⠏⠄⠄⠄⠄⠄⠄⠄⠄⠄⠄⠄⠄⠄⠄⠄⠄⠄⠄⠄⠄⠄⠈⢧⠄⠄⠄⠄⠙⣧⡀⠄⠄⠄⠄⠄⠄⠄⠄⠄⠄⠄⠄⠄⠄⠄⠄⠄⠄⠄⠄⠄⠄⠄⠄⠄⠄⠄⠄⠄⠄⠄⠄⠄⠄⠄⠄⠄⠄⠄⠄⠄⠄⠄⠄⠄⠄⠄⠄⠄⠄⠄⠄
   // │⠄⠄⠄⠄⠄⠄⠄⢀⠞⠄⠄⠄⠄⠄⢀⣼⠃⠄⠄⠄⠄⠄⠄⠄⠄⠄⠄⠄⠄⠄⠄⠄⠄⠄⠄⠄⠄⠄⠄⠄⠈⢧⠄⠄⠄⠄⠘⢷⡀⠄⠄⠄⠄⠄⠄⠄⠄⠄⠄⠄⠄⠄⠄⠄⠄⠄⠄⠄⠄⠄⠄⠄⠄⠄⠄⠄⠄⠄⠄⠄⠄⠄⠄⠄⠄⠄⠄⠄⠄⠄⠄⠄⠄⠄⠄⠄⠄⠄⠄⠄
   // │⠄⠄⠄⠄⠄⠄⢀⡞⠄⠄⠄⠄⠄⢠⡿⠁⠄⠄⠄⠄⠄⠄⠄⠄⠄⠄⠄⠄⠄⠄⠄⠄⠄⠄⠄⠄⠄⠄⠄⠄⠄⠈⢆⠄⠄⠄⠄⠈⢷⡀⠄⠄⠄⠄⠄⠄⠄⠄⠄⠄⠄⠄⠄⠄⠄⠄⠄⠄⠄⠄⠄⠄⠄⠄⠄⠄⠄⠄⠄⠄⠄⠄⠄⠄⠄⠄⠄⠄⠄⠄⠄⠄⠄⠄⠄⠄⠄⠄⠄⠄
   // │⠄⠄⠄⠄⠄⠄⡜⠄⠄⠄⠄⠄⣰⡟⠄⠄⠄⠄⠄⠄⠄⠄⠄⠄⠄⠄⠄⠄⠄⠄⠄⠄⠄⠄⠄⠄⠄⠄⠄⠄⠄⠄⠘⡆⠄⠄⠄⠄⠈⢷⡄⠄⠄⠄⠄⠄⠄⠄⠄⠄⠄⠄⠄⠄⠄⠄⠄⠄⠄⠄⠄⠄⠄⠄⠄⠄⠄⠄⠄⠄⠄⠄⠄⠄⠄⠄⠄⠄⠄⠄⠄⠄⠄⠄⠄⠄⠄⠄⠄⠄
   // │⠄⠄⠄⠄⠄⡼⠁⠄⠄⠄⠄⣴⠏⠄⠄⠄⠄⠄⠄⠄⠄⠄⠄⠄⠄⠄⠄⠄⠄⠄⠄⠄⠄⠄⠄⠄⠄⠄⠄⠄⠄⠄⠄⠘⡄⠄⠄⠄⠄⠈⢻⡀⠄⠄⠄⠄⠄⠄⠄⠄⠄⠄⠄⠄⠄⠄⠄⠄⠄⠄⠄⠄⠄⠄⠄⠄⠄⠄⠄⠄⠄⠄⠄⠄⠄⠄⠄⠄⠄⠄⠄⠄⠄⠄⠄⠄⠄⠄⠄⠄
   // │⠄⠄⠄⠄⡼⠁⠄⠄⠄⢀⡾⠁⠄⠄⠄⠄⠄⠄⠄⠄⠄⠄⠄⠄⠄⠄⠄⠄⠄⠄⠄⠄⠄⠄⠄⠄⠄⠄⠄⠄⠄⠄⠄⠄⠹⡄⠄⠄⠄⠄⠄⢿⡄⠄⠄⠄⠄⠄⠄⠄⠄⠄⠄⠄⠄⠄⠄⠄⠄⠄⠄⠄⠄⠄⠄⠄⠄⠄⠄⠄⠄⠄⠄⠄⠄⠄⠄⠄⠄⠄⠄⠄⠄⠄⠄⠄⠄⠄⠄⠄
   // │⠄⠄⠄⢰⠁⠄⠄⠄⣠⡟⠁⠄⠄⠄⠄⠄⠄⠄⠄⠄⠄⠄⠄⠄⠄⠄⠄⠄⠄⠄⠄⠄⠄⠄⠄⠄⠄⠄⠄⠄⠄⠄⠄⠄⠄⠹⡀⠄⠄⠄⠄⠄⢷⡄⠄⠄⠄⠄⠄⠄⠄⠄⠄⠄⠄⠄⠄⠄⠄⠄⠄⠄⠄⠄⠄⠄⠄⠄⠄⠄⠄⠄⠄⠄⠄⠄⠄⠄⠄⠄⠄⠄⠄⠄⠄⠄⠄⠄⠄⠄
   // │⠄⠄⢠⠇⠄⠄⢀⣰⠟⠄⠄⠄⠄⠄⠄⠄⠄⠄⠄⠄⠄⠄⠄⠄⠄⠄⠄⠄⠄⠄⠄⠄⠄⠄⠄⠄⠄⠄⠄⠄⠄⠄⠄⠄⠄⠄⢳⡀⠄⠄⠄⠄⠈⢷⡀⠄⠄⠄⠄⠄⠄⠄⠄⠄⠄⠄⠄⠄⠄⠄⠄⠄⠄⠄⠄⠄⠄⠄⠄⠄⠄⠄⠄⠄⠄⠄⠄⠄⠄⠄⠄⠄⠄⠄⠄⠄⠄⠄⠄⠄
   // │⠄⢀⠎⠄⠄⣠⡾⠃⠄⠄⠄⠄⠄⠄⠄⠄⠄⠄⠄⠄⠄⠄⠄⠄⠄⠄⠄⠄⠄⠄⠄⠄⠄⠄⠄⠄⠄⠄⠄⠄⠄⠄⠄⠄⠄⠄⠄⢣⠄⠄⠄⠄⠄⠈⢷⡀⠄⠄⠄⠄⠄⠄⠄⠄⠄⠄⠄⠄⠄⠄⠄⠄⠄⠄⠄⠄⠄⠄⠄⠄⠄⠄⠄⠄⠄⠄⠄⠄⠄⠄⠄⠄⠄⠄⠄⠄⠄⠄⠄⠄
   // │⠄⡞⠄⢀⣴⠋⠄⠄⠄⠄⠄⠄⠄⠄⠄⠄⠄⠄⠄⠄⠄⠄⠄⠄⠄⠄⠄⠄⠄⠄⠄⠄⠄⠄⠄⠄⠄⠄⠄⠄⠄⠄⠄⠄⠄⠄⠄⠈⣆⠄⠄⠄⠄⠄⠈⢿⡀⠄⠄⠄⠄⠄⠄⠄⠄⠄⠄⠄⠄⠄⠄⠄⠄⠄⠄⠄⠄⠄⠄⠄⠄⠄⠄⠄⠄⠄⠄⠄⠄⠄⠄⠄⠄⠄⠄⠄⠄⠄⠄⠄
   // │⣜⣠⡾⠋⠄⠄⠄⠄⠄⠄⠄⠄⠄⠄⠄⠄⠄⠄⠄⠄⠄⠄⠄⠄⠄⠄⠄⠄⠄⠄⠄⠄⠄⠄⠄⠄⠄⠄⠄⠄⠄⠄⠄⠄⠄⠄⠄⠄⠘⡆⠄⠄⠄⠄⠄⠈⣷⡀⠄⠄⠄⠄⠄⠄⠄⠄⠄⠄⠄⠄⠄⠄⠄⠄⠄⠄⠄⠄⠄⠄⠄⠄⠄⠄⠄⠄⠄⠄⠄⠄⠄⠄⠄⠄⠄⠄⠄⠄⠄⡼
   // ┼ ─ ─ ─ ─ ┼ ─ ─ ─ ─ ┼ ─ ─ ─ ─ ┼ ─ ─ ─ ─ ┼ ─ ─ ─ ─ ┼─ ─ ─ ─ ┼ ─ ─ ─ ─ ┼ ─ ─ ─ ─ ┼ ─ ─ ─ ─ ┼ ─ ─ ─ ─ 
   // 0.0     10       20       30       40       50       60       70       80       90      100 s
   // │⠄⠄⠄⠄⠄⠄⠄⠄⠄⠄⠄⠄⠄⠄⠄⠄⠄⠄⠄⠄⠄⠄⠄⠄⠄⠄⠄⠄⠄⠄⠄⠄⠄⠄⠄⠄⠄⠄⠄⠄⠄⠄⠄⠄⠄⠄⠄⠄⠄⠄⠄⢧⠄⠄⠄⠄⠄⠄⠘⣧⡀⠄⠄⠄⠄⠄⠄⠄⠄⠄⠄⠄⠄⠄⠄⠄⠄⠄⠄⠄⠄⠄⠄⠄⠄⠄⠄⠄⠄⠄⠄⠄⠄⠄⠄⠄⢠⠏⠄⠄
   // │⠄⠄⠄⠄⠄⠄⠄⠄⠄⠄⠄⠄⠄⠄⠄⠄⠄⠄⠄⠄⠄⠄⠄⠄⠄⠄⠄⠄⠄⠄⠄⠄⠄⠄⠄⠄⠄⠄⠄⠄⠄⠄⠄⠄⠄⠄⠄⠄⠄⠄⠄⠈⢇⠄⠄⠄⠄⠄⠄⠘⣧⠄⠄⠄⠄⠄⠄⠄⠄⠄⠄⠄⠄⠄⠄⠄⠄⠄⠄⠄⠄⠄⠄⠄⠄⠄⠄⠄⠄⠄⠄⠄⠄⠄⠄⠄⡎⠄⠄⠄
   // │⠄⠄⠄⠄⠄⠄⠄⠄⠄⠄⠄⠄⠄⠄⠄⠄⠄⠄⠄⠄⠄⠄⠄⠄⠄⠄⠄⠄⠄⠄⠄⠄⠄⠄⠄⠄⠄⠄⠄⠄⠄⠄⠄⠄⠄⠄⠄⠄⠄⠄⠄⠄⠘⣆⠄⠄⠄⠄⠄⠄⠘⣦⠄⠄⠄⠄⠄⠄⠄⠄⠄⠄⠄⠄⠄⠄⠄⠄⠄⠄⠄⠄⠄⠄⠄⠄⠄⠄⠄⠄⠄⠄⠄⠄⠄⡞⠄⠄⠄⠄
   // │⠄⠄⠄⠄⠄⠄⠄⠄⠄⠄⠄⠄⠄⠄⠄⠄⠄⠄⠄⠄⠄⠄⠄⠄⠄⠄⠄⠄⠄⠄⠄⠄⠄⠄⠄⠄⠄⠄⠄⠄⠄⠄⠄⠄⠄⠄⠄⠄⠄⠄⠄⠄⠄⠘⡄⠄⠄⠄⠄⠄⠄⠙⣇⠄⠄⠄⠄⠄⠄⠄⠄⠄⠄⠄⠄⠄⠄⠄⠄⠄⠄⠄⠄⠄⠄⠄⠄⠄⠄⠄⠄⠄⠄⠄⡼⠄⠄⠄⠄⠄
   // │⠄⠄⠄⠄⠄⠄⠄⠄⠄⠄⠄⠄⠄⠄⠄⠄⠄⠄⠄⠄⠄⠄⠄⠄⠄⠄⠄⠄⠄⠄⠄⠄⠄⠄⠄⠄⠄⠄⠄⠄⠄⠄⠄⠄⠄⠄⠄⠄⠄⠄⠄⠄⠄⠄⠹⡀⠄⠄⠄⠄⠄⠄⠸⣧⠄⠄⠄⠄⠄⠄⠄⠄⠄⠄⠄⠄⠄⠄⠄⠄⠄⠄⠄⠄⠄⠄⠄⠄⠄⠄⠄⠄⠄⣰⠁⠄⠄⠄⠄⢠
   // │⠄⠄⠄⠄⠄⠄⠄⠄⠄⠄⠄⠄⠄⠄⠄⠄⠄⠄⠄⠄⠄⠄⠄⠄⠄⠄⠄⠄⠄⠄⠄⠄⠄⠄⠄⠄⠄⠄⠄⠄⠄⠄⠄⠄⠄⠄⠄⠄⠄⠄⠄⠄⠄⠄⠄⠹⡀⠄⠄⠄⠄⠄⠄⠘⣧⠄⠄⠄⠄⠄⠄⠄⠄⠄⠄⠄⠄⠄⠄⠄⠄⠄⠄⠄⠄⠄⠄⠄⠄⠄⠄⠄⢰⠃⠄⠄⠄⠄⢀⡿
   // │⠄⠄⠄⠄⠄⠄⠄⠄⠄⠄⠄⠄⠄⠄⠄⠄⠄⠄⠄⠄⠄⠄⠄⠄⠄⠄⠄⠄⠄⠄⠄⠄⠄⠄⠄⠄⠄⠄⠄⠄⠄⠄⠄⠄⠄⠄⠄⠄⠄⠄⠄⠄⠄⠄⠄⠄⢳⡀⠄⠄⠄⠄⠄⠄⠙⣧⡀⠄⠄⠄⠄⠄⠄⠄⠄⠄⠄⠄⠄⠄⠄⠄⠄⠄⠄⠄⠄⠄⠄⠄⠄⣠⠃⠄⠄⠄⠄⢠⡿⠁
   // │⠄⠄⠄⠄⠄⠄⠄⠄⠄⠄⠄⠄⠄⠄⠄⠄⠄⠄⠄⠄⠄⠄⠄⠄⠄⠄⠄⠄⠄⠄⠄⠄⠄⠄⠄⠄⠄⠄⠄⠄⠄⠄⠄⠄⠄⠄⠄⠄⠄⠄⠄⠄⠄⠄⠄⠄⠄⢳⠄⠄⠄⠄⠄⠄⠄⠘⢷⡀⠄⠄⠄⠄⠄⠄⠄⠄⠄⠄⠄⠄⠄⠄⠄⠄⠄⠄⠄⠄⠄⠄⢠⠃⠄⠄⠄⠄⢰⡟⠄⠄
   // │⠄⠄⠄⠄⠄⠄⠄⠄⠄⠄⠄⠄⠄⠄⠄⠄⠄⠄⠄⠄⠄⠄⠄⠄⠄⠄⠄⠄⠄⠄⠄⠄⠄⠄⠄⠄⠄⠄⠄⠄⠄⠄⠄⠄⠄⠄⠄⠄⠄⠄⠄⠄⠄⠄⠄⠄⠄⠄⢳⠄⠄⠄⠄⠄⠄⠄⠈⢳⡄⠄⠄⠄⠄⠄⠄⠄⠄⠄⠄⠄⠄⠄⠄⠄⠄⠄⠄⠄⠄⢠⠎⠄⠄⠄⠄⣰⠏⠄⠄⠄
   // │⠄⠄⠄⠄⠄⠄⠄⠄⠄⠄⠄⠄⠄⠄⠄⠄⠄⠄⠄⠄⠄⠄⠄⠄⠄⠄⠄⠄⠄⠄⠄⠄⠄⠄⠄⠄⠄⠄⠄⠄⠄⠄⠄⠄⠄⠄⠄⠄⠄⠄⠄⠄⠄⠄⠄⠄⠄⠄⠄⢣⠄⠄⠄⠄⠄⠄⠄⠄⢿⡄⠄⠄⠄⠄⠄⠄⠄⠄⠄⠄⠄⠄⠄⠄⠄⠄⠄⠄⢀⠏⠄⠄⠄⢀⣴⠋⠄⠄⠄⠄
   // │⠄⠄⠄⠄⠄⠄⠄⠄⠄⠄⠄⠄⠄⠄⠄⠄⠄⠄⠄⠄⠄⠄⠄⠄⠄⠄⠄⠄⠄⠄⠄⠄⠄⠄⠄⠄⠄⠄⠄⠄⠄⠄⠄⠄⠄⠄⠄⠄⠄⠄⠄⠄⠄⠄⠄⠄⠄⠄⠄⠄⢣←--   τ   -→⠹⣦⠄⠄⠄⠄⠄⠄⠄⠄⠄⠄⠄⠄⠄⠄⠄⠄⢠⠋⠄⠄⠄⢠⡾⠁⠄⠄⠄⠄⠄
   // │⠄⠄⠄⠄⠄⠄⠄⠄⠄⠄⠄⠄⠄⠄⠄⠄⠄⠄⠄⠄⠄⠄⠄⠄⠄⠄⠄⠄⠄⠄⠄⠄⠄⠄⠄⠄⠄⠄⠄⠄⠄⠄⠄⠄⠄⠄⠄⠄⠄⠄⠄⠄⠄⠄⠄⠄⠄⠄⠄⠄⠄⠳⡀⠄⠄⠄⠄⠄⠄⠄⠈⢷⡄⠄⠄⠄⠄⠄⠄⠄⠄⠄⠄⠄⠄⠄⢠⠃⠄⠄⠄⣴⠏⠄⠄⠄⠄⠄⠄⠄
   // │⠄⠄⠄⠄⠄⠄⠄⠄⠄⠄⠄⠄⠄⠄⠄⠄⠄⠄⠄⠄⠄⠄⠄⠄⠄⠄⠄⠄⠄⠄⠄⠄⠄⠄⠄⠄⠄⠄⠄⠄⠄⠄⠄⠄⠄⠄⠄⠄⠄⠄⠄⠄⠄⠄⠄⠄⠄⠄⠄⠄⠄⠄⠱⡄⠄⠄⠄⠄⠄⠄⠄⠄⠹⢦⣀⠄⠄⠄⠄⠄⠄⠄⠄⠄⠄⡠⠃⠄⠄⣠⠞⠁⠄⠄⠄⠄⠄⠄⠄⠄
   // │⠄⠄⠄⠄⠄⠄⠄⠄⠄⠄⠄⠄⠄⠄⠄⠄⠄⠄⠄⠄⠄⠄⠄⠄⠄⠄⠄⠄⠄⠄⠄⠄⠄⠄⠄⠄⠄⠄⠄⠄⠄⠄⠄⠄⠄⠄⠄⠄⠄⠄⠄⠄⠄⠄⠄⠄⠄⠄⠄⠄⠄⠄⠄⠙⣄⠄⠄⠄⠄⠄⠄⠄⠄⠈⠙⢶⣄⠄⠄⠄⠄⠄⠄⢀⡔⠁⢀⣠⠞⠁⠄⠄⠄⠄⠄⠄⠄⠄⠄⠄
   // │⠄⠄⠄⠄⠄⠄⠄⠄⠄⠄⠄⠄⠄⠄⠄⠄⠄⠄⠄⠄⠄⠄⠄⠄⠄⠄⠄⠄⠄⠄⠄⠄⠄⠄⠄⠄⠄⠄⠄⠄⠄⠄⠄⠄⠄⠄⠄⠄⠄⠄⠄⠄⠄⠄⠄⠄⠄⠄⠄⠄⠄⠄⠄⠄⠈⠳⡀⠄⠄⠄⠄⠄⠄⠄⠄⠄⠉⠻⠶⣤⣄⣀⣠⣮⡴⠶⠋⠁⠄⠄⠄⠄⠄⠄⠄⠄⠄⠄⠄⠄
   // │⠄⠄⠄⠄⠄⠄⠄⠄⠄⠄⠄⠄⠄⠄⠄⠄⠄⠄⠄⠄⠄⠄⠄⠄⠄⠄⠄⠄⠄⠄⠄⠄⠄⠄⠄⠄⠄⠄⠄⠄⠄⠄⠄⠄⠄⠄⠄⠄⠄⠄⠄⠄⠄⠄⠄⠄⠄⠄⠄⠄⠄⠄⠄⠄⠄⠄⠙⢆⡀⠄⠄⠄⠄⠄⠄⠄⠄⠄⠄⠄⢀⠞⠉⠄⠄⠄⠄⠄⠄⠄⠄⠄⠄⠄⠄⠄⠄⠄⠄⠄
   // │⠄⠄⠄⠄⠄⠄⠄⠄⠄⠄⠄⠄⠄⠄⠄⠄⠄⠄⠄⠄⠄⠄⠄⠄⠄⠄⠄⠄⠄⠄⠄⠄⠄⠄⠄⠄⠄⠄⠄⠄⠄⠄⠄⠄⠄⠄⠄⠄⠄⠄⠄⠄⠄⠄⠄⠄⠄⠄⠄⠄⠄⠄⠄⠄⠄⠄⠄⠄⠙⠢⣄⠄⠄⠄⠄⠄⠄⢀⡠⠞⠁⠄⠄⠄⠄⠄⠄⠄⠄⠄⠄⠄⠄⠄⠄⠄⠄⠄⠄⠄
   // │⠄⠄⠄⠄⠄⠄⠄⠄⠄⠄⠄⠄⠄⠄⠄⠄⠄⠄⠄⠄⠄⠄⠄⠄⠄⠄⠄⠄⠄⠄⠄⠄⠄⠄⠄⠄⠄⠄⠄⠄⠄⠄⠄⠄⠄⠄⠄⠄⠄⠄⠄⠄⠄⠄⠄⠄⠄⠄⠄⠄⠄⠄⠄⠄⠄⠄⠄⠄⠄⠄⠄⠉⠓⠒⠒⠒⠋⠁⠄⠄⠄⠄⠄⠄⠄⠄⠄⠄⠄⠄⠄⠄⠄⠄⠄⠄⠄⠄⠄⠄
   // 
   //    Increasing τ gives a slower response.
   // 
   //    Output follows input with a lag = τ   Time to reach steady state = 5τ
   // 
   // 
   // 
   // ▂▂▂▂▂▂▂▂▂▂▂▂▂▂▂▂▂▂▂▂▂▂▂▂▂▂▂▂▂▂▂▂▂▂▂▂▂▂▂▂▂▂▂▂
   // 2.5      Operating modes
   // 
   // 
   // The block supports two modes of operation:
   // 
   //    •   Automatic mode:
   //      The module automatically calculates the elapsed time since the simulation started 
   //      and generates the appropriate output value for any form of input.
   // 
   //      Automatic mode can accommodate any form of input (step, ramp, sinusoid, 
   //      freeform &c.).
   // 
   //    •   Manual mode:
   //      The current elapsed time and fixed input value is supplied manually to the module; 
   //      the module will then calculate the output value based on a step input at this input 
   //      value and at this time value.
   // 
   //      Manual mode only supports a step form of input (the input is considered to be a step 
   //      input that changed to the manually specified input value at time = 0, and that prior to 
   //      this the input was zero. I.e. a step input that changed from zero to the specified value 
   //      at time = 0).
   // 
   // 
   //                ━━━   ⬙⬙⬙⬙⬙⬙   ━━━
END_REGION

REGION Network 2: Block description — Section 3
   // ▄▄▄▄▄▄▄▄▄▄▄▄▄▄▄▄▄▄▄▄▄▄▄▄▄▄▄▄▄▄▄▄▄▄▄▄▄▄▄▄▄▄▄▄
   // 3.     DETAILED BLOCK DESCRIPTION
   // 
   // 
   // This module, FC19511_StdDebugInst1Order uses user data types to provide the primary 
   // interface to the block. There are four formal parameters:
   // 
   //  ――――――――――――――――――――――――――――――――――――――――――
   //  PARAM         FUNCTION                    TYPE      IN-OUT 
   //  ――――――――――――――――――――――――――――――――――――――――――
   //  SYS_SIGNALS      Common system signals              UT21000    In
   //           logic and timing signals for parametric access
   // 
   //  TRIGGER       Activates the simulation (the simulation will run     Bool      In
   //           whilever this signal is high), the elapsed time 
   //           is measured from the rising edge of this signal
   // 
   //  INPUT        The input time function, x(t) in the calculations     Real      In
   // 
   //  DYNAMIC_DATA      Data structure that holds the live data for the       UT39512    InOut
   //           simulation (damping factor, natural frequency, 
   //           system gain, elapsed time &c.)
   // 
   //  OUTPUT       The output time response, y(t) in the calculations   Real      Out
   //  ――――――――――――――――――――――――――――――――――――――――――
   // 
   // The DYNAMIC_DATA parameter is a UDT that holds all the data for the simulation.
   // 
   //  ――――――――――――――――――――――――――――――――――――――――――
   //  PARAM         ASSOCIATED UDT          ASSOCIATED DATA BLOCK
   //  ――――――――――――――――――――――――――――――――――――――――――
   //  DYNAMIC_DATA   UT39511_Dy_DebugInst1Order      DB39511_Dy_DebugInst1Order
   //  ――――――――――――――――――――――――――――――――――――――――――
   // 
   // 
   // Section 6 contains a full list of all variables within these UDTs.
   // 
   // 
   // 
   // ▂▂▂▂▂▂▂▂▂▂▂▂▂▂▂▂▂▂▂▂▂▂▂▂▂▂▂▂▂▂▂▂▂▂▂▂▂▂▂▂▂▂▂▂
   // 3.1      The primary simulation signals
   // 
   // 
   // The simulation is based upon various signals passed to the module and the elapsed time since 
   // the simulation started:
   // 
   //  ――――――――――――――――――――――――――――――――――――――――――
   //  SIGNAL         FUNCTION               RANGE       ACCESSED VIA
   //  ――――――――――――――――――――――――――――――――――――――――――
   //  INPUT         The INPUT parameter is the x value    Unrestricted     Parameter 
   //            in the calculations of § 3.2
   // 	
   //  OUTPUT        The OUTPUT parameter is the y value   Unrestricted     Parameter 
   //            in the calculations of § 3.2
   // 
   //  TRIGGER        The TRIGGER parameter activates      0 or 1     Parameter
   //            the simulation
   // 
   //  k_Gain          The system gain (K) term         Unrestricted     UT39511
   //            in the calculations of § 3.2       typ. 1-10
   // 
   //  k_TimeConstant     The system time constant (τ) term in   +ve number      UT39511
   //            the calculations of § 3.2.
   //            In units of seconds (s)
   // 
   //  actual_PrevOutput   The resulting output calculated in the  Unrestricted     UT39511
   //            previous iteration of the calculation
   // 
   //  actual_StartTime   The CPU time when the simulation    DTL value    UT39511
   //            started (rising edge of TRIGGER)      of RTC
   // 
   //  actual_Time      The current CPU time, for the current    DTL value    UT39511
   //            iteration of the calculation         of RTC
   //            (time at y[n])
   // 
   //  actual_PrevTime    The CPU time of the last iteration    DTL value    UT39511
   //            of the calculation              of RTC
   //            (time at y[n-1])
   // 
   //  actual_RunTime     The elapsed time of the simulation      +ve number      UT39511
   //            in seconds (s)              calculated by
   //                              the module
   // 
   //  actual_DeltaTime     Time between the current iteration      +ve number      UT39511
   //            and the previous iteration, Δt in the     calculated by 
   //            calculations:             the module
   //            = actual_Time – actual_PrevTime
   //            In units of seconds (s)
   //  ――――――――――――――――――――――――――――――――――――――――――
   // 
   // 
   // The system time constant (k_TimeConstant), determines the lag of the system, the higher the 
   // value, the slower the response.
   // 
   // The system gain (k_Gain), is simply a common multiplier that amplifies the output response. 
   // By default the system gain is set to a value of one (i.e. unity gain).
   // 
   // The elapsed time actual_RunTime is calculated from the real time clock within the CPU. On the 
   // rising edge of the TRIGGER parameter, the CPU real time clock is read and the value stored in 
   // the variable actual_StartTime, on each subsequent call to the block, the real time clock is 
   // once again read and stored in the variable actual_Time. The elapsed time is calculated by 
   // subtracting the actual_StartTime value from the actual_Time value and converting the result 
   // to seconds this is then stored as the actual_RunTime value.
   // 
   // The TRIGGER signal is simply used to start and stop the simulation. A rising edge on the 
   // TRIGGER signal causes the current CPU time to be stored (actual_StartTime) and sets the 
   // elapsed time to zero (actual_RunTime). The simulation will run whilever the TRIGGER signal is 
   // high (has a value of 1), each time the module is called, the elapsed time (actual_RunTime) is 
   // updated (see the previous paragraph) and the output calculated accordingly.
   // 
   // If the simulation is active (the TRIGGER signal is high, has a value of 1) the time between the 
   // current module call (actual_Time) and the previous module call (actual_PrevTime) is calculated 
   // and stored in the variable actual_DeltaTime (∆t in the calculations), this is calculated as follows:
   // 
   //      actual_DeltaTime= actual_Time-actual_PrevTime
   // 
   // At the end of the current module call, the actual_PrevTime is set to the actual_Time, for the 
   // next iteration of the calculation.
   // 
   // At the end of the current module call, the actual_PrevOutput is set to the OUTPUT, value for the 
   // next iteration of the calculation.
   // 
   // If the TRIGGER signal is low (0), the simulation is instantly stopped and the OUTPUT parameter is 
   // set to zero.
   // 
   // 
   // 
   // ▂▂▂▂▂▂▂▂▂▂▂▂▂▂▂▂▂▂▂▂▂▂▂▂▂▂▂▂▂▂▂▂▂▂▂▂▂▂▂▂▂▂▂▂
   // 3.2      The response calculation
   // 
   // 
   // Two forms of calculation are carried out by the module, the first is the iterative, real-time 
   // calculation for the automatic response, this is given in equation (2.2). The second is the discrete 
   // manual response calculation given in equation (2.3). These are reproduced below.
   // 
   // The calculations below use Greek characters for the main variables, the calculations use various 
   // parameters and UDT variables that have plain English names, The association between these 
   // variables and the Greek nomenclature is given below.
   // 
   // 
   // ――――――――――――――――――――――――――――――――――――――――――――――――
   // REAL-TIME AUTOMATIC SIMULATION         from equation 2.2
   // 
   //    y[n] = Ka x[n]  ┼ (1-a) y[n-1]  (3.1)
   // 
   //              ΔT
   //    where:   a = ----------
   //            τ+ΔT
   // ――――――――――――――――――――――――――――――――――――――――――――――――
   // DISCRETE MANUAL RESPONSE TO A STEP INPUT      from equation 2.3
   // 
   //          ┌      -t/τ  ┐
   //    y(t) = KX│ 1 ─  e   │    (3.2)
   //          └       ┘
   // ――――――――――――――――――――――――――――――――――――――――――――――――
   // Where:    K      is the system gain (a constant number)             k_Gain
   //      τ      is the system time constant (in seconds)             k_TimeConstant
   //      Δt    is the sampling interval between calculations (in seconds)  actual_DeltaTime
   //      X/x[n] is the input at the current iteration or in manual mode    parameter INPUT
   //      y/y[n]  is the output at the current iteration or in manual mode    parameter OUTPUT
   //      y[n-1] is the output at the previous iteration             actual_PrevOutput
   // 
   // Note:    If the system gain k_Gain is set zero, the OUTPUT will be zero under all circumstances.
   // 
   // Each of these calculations can be accommodated with the mathematical functions available to a 
   // Siemens Controller, see § 3.4.
   // 
   // 
   // 
   // 
   // ▂▂▂▂▂▂▂▂▂▂▂▂▂▂▂▂▂▂▂▂▂▂▂▂▂▂▂▂▂▂▂▂▂▂▂▂▂▂▂▂▂▂▂▂
   // 3.3      Status and informative signals
   // 
   // 
   // The module produces various status signals that reflect the nature of the simulation:
   // 
   //  DATA STRUCTURE      UT39511_Dy_DebugInst1Order
   //  ――――――――――――――――――――――――――――――――――――――――――
   //  SIGNAL           FUNCTION            TYPE   DETAILS
   //  ――――――――――――――――――――――――――――――――――――――――――
   //  status_Running        The simulation is running     Bool    1 = Simulation is running 
   //                               0 = Simulation is stopped
   // 
   //  status_Stopped       The simulation is stopped    Bool    1 = Simulation is stopped 
   //                               0 = Simulation is running
   // 
   //  status_SteadyState      Simulation has achieved   Bool    1 = Stady state achieved
   //                 steady state ±2%           0 = Not in steady state
   // 
   //  cal_TimeSteady       Time to reach steady state      Real Seconds
   // 
   // 
   //  ――――――――――――――――――――――――――――――――――――――――――
   // 
   // The status_Running and status_Stopped are determined purely by the status of the TRIGGER 
   // parameter, if this is set high (1), status_Running will be high and status_Stopped low. If  TRIGGER 
   // parameter, if this is set low (0), status_Running will be low and status_Stopped high. The 
   // status_Running and status_Stopped signals are always the inverse of each other.
   // 
   // If the simulation has reached a steady state, i.e. the non-linear relationship between the output 
   // and the input that occurs at the start of the simulation has concluded, the status_SteadyState 
   // signal will be set high (1), it will be low (0) until the steady state conditions are achieved 
   // (typically, this is at 5×τ seconds after the start of the simulation).
   // 
   // In addition, the variable cal_TimeSteady give the time at which the steady state will be reached 
   // (in seconds), this is true for all forms of input.
   // 
   // 
   // 
   // ▂▂▂▂▂▂▂▂▂▂▂▂▂▂▂▂▂▂▂▂▂▂▂▂▂▂▂▂▂▂▂▂▂▂▂▂▂▂▂▂▂▂▂▂
   // 3.4     Expressing the calculations in Controller operations
   // 
   // The calculations above must be rendered in a form suitable for the Simatic S7-1500 Controller, 
   // using the mathematical operations available to that Controller, these are listed in Table 2.1.
   // 
   // To perform the calculations in the Controller it will be necessary to use partial calculation to 
   // hold separate components of the overall calculation and combine these to produce the final 
   // result. 
   // 
   // The following sections breakdown each of the response calculations into these partial 
   // calculations and demonstrate how these are then combined to provide a final result that is 
   // compatible with the Controller mathematical operations and Controller notations.
   // 
   // 
   // 
   // ▁▁▁▁▁▁▁▁▁▁▁▁▁▁▁▁▁▁▁▁▁▁▁▁▁▁▁▁▁▁▁▁▁▁▁▁▁▁▁▁▁▁▁▁
   // 3.4.1     Real-time simulation calculation
   // 
   // 
   // CALCULATION:
   //                               ΔT
   //    y[n] = Ka x[n]  ┼ (1-a) y[n-1]   where: a = ----------
   //                             τ+ΔT
   // 
   // Is rendered into the correct format as follows:
   // 
   // 
   //  cal_01 = ΔT             =  actual_Time - actual_PrevTime
   // 
   //  cal_02 = τ + ΔT             = k_TimeConstant + cal_01
   // 
   //                ΔT
   //  cal_03 = a = ----------          = cal_01 ÷ cal_02
   //                 τ+ΔT
   // 
   //  cal_04 = 1 - a             = 1 - cal_03
   // 
   // 
   //  cal_05 = Kax[n]            = k_Gain × cal_03 × INPUT
   // 
   //  cal_06 = (1-a) y[n-1]          = cal_04 × actual_PrevOutput
   // 
   // 
   //  OUTPUT  = Ka x[n]  ┼ (1-a) y[n-1]      = cal_05 × cal_06
   // 
   // 
   // 
   // ▁▁▁▁▁▁▁▁▁▁▁▁▁▁▁▁▁▁▁▁▁▁▁▁▁▁▁▁▁▁▁▁▁▁▁▁▁▁▁▁▁▁▁▁
   // 3.4.2     Discrete manual response to a step input
   // 
   // 
   // CALCULATION:
   // 
   //          ┌      -t/τ  ┐
   //    y(t) = KX│ 1 ─  e   │
   //          └       ┘
   // 
   // 
   // Is rendered into the correct format as follows:
   // 
   // 
   //  cal_01 =  t/τ             = - 1 × actual_RunTime ÷  k_TimeConstant
   // 
   //          - t/τ
   //  cal_02 = ｅ              = EXP (cal_01)
   // 
   //                - t/τ
   //  cal_03 = 1 ─  ｅ              = 1 - cal_02
   // 
   // 
   //              ┌      -t/τ  ┐
   //  OUTPUT  = KX│ 1 ─  e   │       = k_Gain × INPUT × cal_03
   //              └       ┘
   // 
   // 
   // 
   // ▂▂▂▂▂▂▂▂▂▂▂▂▂▂▂▂▂▂▂▂▂▂▂▂▂▂▂▂▂▂▂▂▂▂▂▂▂▂▂▂▂▂▂▂
   // 3.5     Operating modes
   // 
   // 
   // This block FC19511_StdDebugInst1Order supports manual and automatic operating modes, the 
   // default mode is automatic.
   // 
   // The module can be switched between automatic and manual modes with the 
   // mode_AutMan signal:
   // 
   //  DATA STRUCTURE    UT39511_Dy_DebugInst1Order
   //  ――――――――――――――――――――――――――――――――――――――――――
   //  SIGNAL         FUNCTION               TYPE     DETAILS
   //  ――――――――――――――――――――――――――――――――――――――――――
   //  Mode_AutMan     Specifies the operating mode of     Bool  1 = automatic mode
   //            the simulation                 0 = manual mode
   // 
   //  Mode_ManTime     Specifies the manual time value of       Real     Elapsed time
   //            the simulation in seconds           in seconds
   // 
   //  status_Aut      The simulation is in automatic mode   Bool  1 = auto mode
   //                                  0 = not in auto
   // 
   //  status_Man       The simulation is in manual mode    Bool  1 = manual mode
   //                                  0 = not in manual
   //  ――――――――――――――――――――――――――――――――――――――――――  
   // 
   // 
   // 
   // ▁▁▁▁▁▁▁▁▁▁▁▁▁▁▁▁▁▁▁▁▁▁▁▁▁▁▁▁▁▁▁▁▁▁▁▁▁▁▁▁▁▁▁▁
   // 3.5.1    Automatic mode
   // 
   // 
   // By default the module will be in automatic mode. 
   // 
   // In automatic mode, if the simulation is active (TRIGGER = 1), the module carries out the real-time 
   // calculation given in § 3.4.1. 
   // 
   // In automatic mode, a real time simulation occurs, generating responses similar to those shown 
   // in the plots of § 2.4 (depending on the nature of the input).
   //  
   // 
   // 
   // 
   // ▁▁▁▁▁▁▁▁▁▁▁▁▁▁▁▁▁▁▁▁▁▁▁▁▁▁▁▁▁▁▁▁▁▁▁▁▁▁▁▁▁▁▁▁
   // 3.5.2    Manual mode
   // 
   // 
   // In manual mode, if the simulation is active (TRIGGER = 1), the module carries out the discrete 
   // response to a step input calculation given in § 3.4.2. 
   // 
   // The difference with manual mode, is that the time used in the calculation must be uniquely 
   // specified; a manual time value must be provided.
   // 
   // The manual time is given in the variable mode_ManTime and is specified in seconds.
   // 
   // If mode mode_ManTime remains constant between module calls, the module will return the 
   // same OUTPUT value each time (assuming all other signals remain unchanged).
   // 
   // The manual mode response is that of a step input, the value of the INPUT parameter is taken as 
   // the starting value of the step at time = 0.
   // 
   // 
   //                ━━━   ⬙⬙⬙⬙⬙⬙   ━━━
END_REGION

REGION Network 3: Block description — Sections 4 to 10
   // ▄▄▄▄▄▄▄▄▄▄▄▄▄▄▄▄▄▄▄▄▄▄▄▄▄▄▄▄▄▄▄▄▄▄▄▄▄▄▄▄▄▄▄▄
   // 4.     Supervisory system interface
   // 
   // 
   // There is no supervisory system interface for this block. It is a debug simulation module and as 
   // such has no graphical symbol, block icon or faceplate.
   // 
   // 
   //                ━━━   ⬙⬙⬙⬙⬙⬙   ━━━
   // 
   // 
   // 
   // ▄▄▄▄▄▄▄▄▄▄▄▄▄▄▄▄▄▄▄▄▄▄▄▄▄▄▄▄▄▄▄▄▄▄▄▄▄▄▄▄▄▄▄▄
   // 5.     PARAMETERS
   // 
   // 
   // The following parameters are associated with the block:
   // 
   //  
   //  ――――――――――――――――――――――――――――――――――――――――――
   //  PARAM         FUNCTION                    TYPE      IN-OUT 
   //  ――――――――――――――――――――――――――――――――――――――――――
   //  SYS_SIGNALS      Common system signals              UT21000    In
   //           logic and timing signals for parametric access
   // 
   //  TRIGGER       Activates the simulation (the simulation will run     Bool      In
   //           whilever this signal is high), the elapsed time 
   //           is measured from the rising edge of this signal
   // 
   //  INPUT        The input time function, x(t) in the calculations     Real      In
   // 
   //  DYNAMIC_DATA      Data structure that holds the live data for the       UT39511    InOut
   //           simulation (damping factor, natural frequency, 
   //           system gain, elapsed time &c.)
   // 
   //  OUTPUT       The output time response, y(t) in the calculations   Real      Out
   //  ――――――――――――――――――――――――――――――――――――――――――
   // 
   //                ━━━   ⬙⬙⬙⬙⬙⬙   ━━━
   // 
   // 
   // 
   // ▄▄▄▄▄▄▄▄▄▄▄▄▄▄▄▄▄▄▄▄▄▄▄▄▄▄▄▄▄▄▄▄▄▄▄▄▄▄▄▄▄▄▄▄
   // 6.     DATA STRUCTURES AND USAGE
   // 
   // 
   // The block has the following associated data structure:
   // 
   // 
   //  ――――――――――――――――――――――――――――――――――――――――――
   //  DATA STRUCTURE             DESCRIPTION
   //  ――――――――――――――――――――――――――――――――――――――――――
   //  UT01000_St_SysRevision          Revision information for this block    See FC01001
   //  UT01001_St_SysLicence           Licence information for this block  See FC01001
   //  UT21000_Dy_SysSignals           System signals for logic and timing  See FC01001
   // 
   //  UT39511_Dy_DebugInst1Order        Dynamic data storage, contains live data, such as 
   //                     calculation variables, elapsed time, oscillation 
   //                     frequency and status signals
   //  ――――――――――――――――――――――――――――――――――――――――――
   // 
   // 
   // ▂▂▂▂▂▂▂▂▂▂▂▂▂▂▂▂▂▂▂▂▂▂▂▂▂▂▂▂▂▂▂▂▂▂▂▂▂▂▂▂▂▂▂▂
   // 6.1      UT39511_Dy_DebugInst1Order
   // 
   // The static data structure for an isolating valve.
   // 
   // 
   // 
   //  UT39511_Dy_DebugInst1Order (full contents)
   //  ――――――――――――――――――――――――――――――――――――――――――
   //  SIGNAL NAME          FUNCTION                     TYPE
   //  ――――――――――――――――――――――――――――――――――――――――――
   //  k_Gain             CONSTANT — Simulation system gain        Real
   //  k_TimeConstant        CONSTANT — The system time constant τ (s)       Real
   // 
   //  status_Running      STATUS — Simulation is running  Bool
   //                      (1 = running, 0 = stopped)
   //  status_Stopped        STATUS — Simulation is stopped (not running)    Bool
   //                      (1 = stopped, 0 = running)
   //  status_SteadyState     STATUS — Response is at steady state value             Bool
   //                      (1 = stead state reached ±2%)
   //  status_Aut           STATUS — Simulation is in automatic mode      Bool
   //                      (1 = automatic, 0 = manual)
   //  status_Man          STATUS — Simulation is in manual mode        Bool
   //                      (1 = manual, 0 = automatic)
   // 
   //  cal_TimeSteady        CALC — Time to reach steady state (s)       Real
   //                    zero for unstable response
   // 
   //  mode_AutMan       MODE — Automatic/manual mode selection     Bool
   //                      (1 = auto mode, 0 = manual mode)
   //  mode_ManTime       MODE — Manual mode time value (s)        Real
   // 
   //  actual_Output       ACTUAL — Output signal, same as OUTPUT param    Real
   //                      (y(t) or y[n])
   //  actual_PrevOutput      ACTUAL — Output value from the previous iteration    Real
   //                      (y[n-1])
   //  actual_StartTime         ACTUAL — CPU time when simulation started       DTL
   //  actual_Time        ACTUAL — CPU time of this iteration of simulation  DTL
   //  actual_PrevTime       ACTUAL — CPU time of last iteration of simulation     DTL
   //  actual_RunTime        ACTUAL — Elapsed time since the            Real
   //                      simulation started (s)
   //  actual_DeltaTime        ACTUAL — Time between this and last iteration (s)   Real
   //  ――――――――――――――――――――――――――――――――――――――――――
   // 
   // 
   //                ━━━   ⬙⬙⬙⬙⬙⬙   ━━━
   // 
   // 
   // 
   // ▄▄▄▄▄▄▄▄▄▄▄▄▄▄▄▄▄▄▄▄▄▄▄▄▄▄▄▄▄▄▄▄▄▄▄▄▄▄▄▄▄▄▄▄
   // 7.     CONSTANTS AND TEMPORARY (LOCAL) DATA
   // 
   // 
   // 
   // ▂▂▂▂▂▂▂▂▂▂▂▂▂▂▂▂▂▂▂▂▂▂▂▂▂▂▂▂▂▂▂▂▂▂▂▂▂▂▂▂▂▂▂▂
   // 7.1     Constants
   // 
   // 
   // The following constants data is used:
   // 
   //  ――――――――――――――――――――――――――――――――――――――――――
   //  SIGNAL NAME       Value     FUNCTION                 TYPE
   //  ――――――――――――――――――――――――――――――――――――――――――
   //  k_NEG_MAX       3.4E-38    Largest negative REAL number         Real
   //  ――――――――――――――――――――――――――――――――――――――――――
   // 
   // 
   // 
   // ▂▂▂▂▂▂▂▂▂▂▂▂▂▂▂▂▂▂▂▂▂▂▂▂▂▂▂▂▂▂▂▂▂▂▂▂▂▂▂▂▂▂▂▂
   // 7.2     Temporary (local) data
   // 
   // 
   // The following temporary data is used:
   // 
   //  ――――――――――――――――――――――――――――――――――――――――――
   //  SIGNAL NAME          FUNCTION                  TYPE
   //  ――――――――――――――――――――――――――――――――――――――――――
   //  revInfo             Revision information for the block         UT01000
   //  licInfo           Licensing information for the block      UT01001
   //  act_CPUTime           Current CPU time (this block call)       DTL
   //  cal_01          Partial calculation see § 3.4 for details      Real
   //  cal_02          Partial calculation see § 3.4 for details      Real
   //  cal_03          Partial calculation see § 3.4 for details      Real
   //  cal_04          Partial calculation see § 3.4 for details      Real
   //  cal_05          Partial calculation see § 3.4 for details      Real
   //  cal_06          Partial calculation see § 3.4 for details      Real
   //  wrkElapsedTime          Working storage area (current elapsed time)    LTIme
   //  wrkDeltaTime         Working storage area (current delta time)   LTIme
   //  wrkInt           Working storage area (integer)          Int
   //  wrkLInt            Working storage area (long integer)        ULInt
   //  wrkReal           Working storage (Real)             Real
   //  ――――――――――――――――――――――――――――――――――――――――――
   // 
   // 
   //                ━━━   ⬙⬙⬙⬙⬙⬙   ━━━
   // 
   // 
   // 
   // ▄▄▄▄▄▄▄▄▄▄▄▄▄▄▄▄▄▄▄▄▄▄▄▄▄▄▄▄▄▄▄▄▄▄▄▄▄▄▄▄▄▄▄▄
   // 8.     BLOCK CALLS AND ASSOCIATIONS
   // 
   // 
   // This section details any blocks which may be called from within this software module (subroutine 
   // functions for example), any partner blocks with which it may be associated (for example a 
   // receive module that is partner with a transmit module &c.). It lists any system functions which 
   // may be called (e.g. reading the real time clock) and any system data types that may be used.
   // 
   // Finally, it lists any special calling requirements for the block (for example, must be called from 
   // within a cyclic interrupt organisation block) and if the block is using “optimised access” (this is 
   // the default arrangement).
   // 
   // 
   // 
   // ▂▂▂▂▂▂▂▂▂▂▂▂▂▂▂▂▂▂▂▂▂▂▂▂▂▂▂▂▂▂▂▂▂▂▂▂▂▂▂▂▂▂▂▂
   // 8.1     Block calls from within this module
   // 
   // 
   // There are no PAL block calls from within this block.
   // 
   // 
   // 
   // ▂▂▂▂▂▂▂▂▂▂▂▂▂▂▂▂▂▂▂▂▂▂▂▂▂▂▂▂▂▂▂▂▂▂▂▂▂▂▂▂▂▂▂▂
   // 8.2     Blocks associated with this module
   // 
   // 
   // This is a stand-alone block and is not associated with any other blocks.
   // 
   // 
   // 
   // ▂▂▂▂▂▂▂▂▂▂▂▂▂▂▂▂▂▂▂▂▂▂▂▂▂▂▂▂▂▂▂▂▂▂▂▂▂▂▂▂▂▂▂▂
   // 8.3     System block calls and system data types
   // 
   // The following calls are made to system blocks:
   // 
   // 
   //  System block calls
   //  ――――――――――――――――――――――――――――――――――――――――――
   //  BLOCK          TITLE             DESCRIPTION  
   //  ――――――――――――――――――――――――――――――――――――――――――
   //  RD_LOC_T             Read the local RTC time    Reads the CPU real time clock 
   //  ――――――――――――――――――――――――――――――――――――――――――
   // 
   // There are no special system data types used.
   // 
   // 
   //                ━━━   ⬙⬙⬙⬙⬙⬙   ━━━
   // 
   // 
   // 
   // ▂▂▂▂▂▂▂▂▂▂▂▂▂▂▂▂▂▂▂▂▂▂▂▂▂▂▂▂▂▂▂▂▂▂▂▂▂▂▂▂▂▂▂▂
   // 8.4     Special properties and requirements
   // 
   // 
   // 
   // ▁▁▁▁▁▁▁▁▁▁▁▁▁▁▁▁▁▁▁▁▁▁▁▁▁▁▁▁▁▁▁▁▁▁▁▁▁▁▁▁▁▁▁▁
   // 8.4.1     Block optimisation, IEC compatibility and library conformance
   // 
   // 
   //    •   Block optimisation is ACTIVE for this block.
   // 
   //    •   The block has been checked for IEC compatibility and is compliant.
   // 
   //    •   The block is compatible with all IEC library-conformance module constraints
   // 
   // 
   // 
   // ▁▁▁▁▁▁▁▁▁▁▁▁▁▁▁▁▁▁▁▁▁▁▁▁▁▁▁▁▁▁▁▁▁▁▁▁▁▁▁▁▁▁▁▁
   // 8.4.2     Calling requirements
   // 
   // 
   // There are no special calling requirements for this block.
   // 
   //                ━━━   ⬙⬙⬙⬙⬙⬙   ━━━
   // 
   // 
   // 
   // ▄▄▄▄▄▄▄▄▄▄▄▄▄▄▄▄▄▄▄▄▄▄▄▄▄▄▄▄▄▄▄▄▄▄▄▄▄▄▄▄▄▄▄▄
   // 9.     EXAMPLE USAGE
   // 
   // 
   // The following shows a typical deployment of FC19512:
   // 
   //                         ┌─────────────
   //      ───────────────────┤ FC19511
   //                         ├───────────────┤
   //    "DB21001_DY_StdGlobalData".SysSignals ─┤ SYS_SIGNALS                  %MD910 
   //                         │               OUTPUT ├─  "SIM001_OUTPUT"
   //                         │               │
   //                                                        "1.0" ─┤ INPUT                     │
   //                         │               │
   //                   %M999.0     │               │
   //                  "SIM001_TRIG" ─┤ TRIGGER                     │
   //                         │               │
   //                         │
   //      "DB39511_Dy_DebugInst1Order".SIM001 ─┤ DYNAMIC_DATA
   //                         │
   //                         │
   //                                         │
   //                                ─────────┘
   // 
   // 
   //               ━━━   ⬙⬙⬙⬙⬙⬙   ━━━
   // 
   // 
   // 
   // ▄▄▄▄▄▄▄▄▄▄▄▄▄▄▄▄▄▄▄▄▄▄▄▄▄▄▄▄▄▄▄▄▄▄▄▄▄▄▄▄▄▄▄▄
   // 10.     TEST AND VERIFICATION PATH
   // 
   // 
   // The following diagram shows the full test and verification path for the formal release of each 
   // version of the software module. See the Test Plan [Ref. 003] for full details, available here:
   //         https://psop.uk/pal-tp-p
   // 
   // 
   //         FC19151-T001
   // 
   //     Test version: 000.801  
   //  Released version: 001.000   
   // Released commit: D0017    
   // 
   //        SCR      SMT 
   // ＿＿＿＿＿＿┌┐＿＿ ▛▜ ＿
   //       └┘   ▙▟  
   // Initial test           
   // 
   // Initial test to release the      
   // module following the      
   // development stage.       
   // Full SMT              
   // 
   // 
   // Where:
   // ――――――――――――――――――――――――――――――――――――――――――――
   //  SCR    Source Code Review      A visual inspection of the software to ensure it has been written  
   // ┌┐             to the correct standards, uses the correct structures within the
   // └┘             software and is generally suitable for deployment.               
   // 
   //  SMT Software Module Test    A full and detailed test of an individual software module in
   //   ▛▜              isolation; such testing requires that all branches of the 
   //   ▙▟              software are tested. 
   // 
   //                It tests all the interfaces to the module, any data recorded or 
   //                stored by the module, all error and exception handling functions 
   //                and tests all timed and interrupt driven operations.
   // 
   //  SCV Software Compatibility     A mechanism for verifying that no executable code software 
   // ╓╖    Verification          changes have been made to a module following changes to
   // ╙╜             comment fields.
   // 
   //                Allows typographical errors &c. to be corrected without forcing 
   //                a full SMT on a module that has not functionally changed.
   // ――――――――――――――――――――――――――――――――――――――――――――
   // 
   // An SCV can only be performed on a module that has at some point previously, successfully 
   // completed both an SCR and SMT. Where an SCV is implemented, it replaces the requirement for 
   // both the SCR and the SMT for the test iteration in question.
   // 
   //                ━━━   ⬙⬙⬙⬙⬙⬙   ━━━
   // 
   // 
   // ██████████████ █ █ █ █  END   █ █ █ █ ██████████████
END_REGION

REGION Network 4: Current revision and modification history
   // ▄▄▄▄▄▄▄▄▄▄▄▄▄▄▄▄▄▄▄▄▄▄▄▄▄▄▄▄▄▄▄▄▄▄▄▄▄▄▄▄▄▄▄▄
   // MODIFICATION HISTORY
   // 
   // 
   // The revision data shown here, in the network comments, contains additional information 
   // reflecting the software development workflow under the version control system (VCS) employed 
   // to track all software changes.
   // 
   // The VCS in use is the Git Source Code Management system in conjunction with the GitHub online 
   // hosting system. The software in its entirety is available in the GitHub remote repository:
   // 
   //      https://github.com/practicalseries/PS2001-pal-software
   // 
   // The repository is public and can be freely copied (forked in GitHub terminology) and used 
   // under the MIT licence. 
   // 
   // The MIT licence is reproduced in full in the last network of this software module.
   // 
   // 
   //  ―――――――――――――――――――――――――――――――――――――――――――
   //  DATE       REVISION             MASTER BRANCH     DEV
   //          (nnn.amm)   COMMIT TAG    (Base ---> Merge)    BRANCH   Author
   //  ———————————————————————————————————————————
   //  2023.02.26    000.101   D0016A-000.101   D0016 N/A     D0016A   M. Gledhill
   //                        FC19511 Block created — Comments added
   //  ———————————————————————————————————————————
   //   Where: nnn  =  Major revision
   //         a  =  Type (1-7 Development, 8 Proving, 9 Qualification, 0 Release)
   //       mm  =  Minor revision (must be 00 if a = 0)
   //         Block properties version number should be set to nn.a (only one decimal place)
   // 
   // ▄▄▄▄▄▄▄▄▄▄▄▄▄▄▄▄▄▄▄▄▄▄▄▄▄▄▄▄▄▄▄▄▄▄▄▄▄▄▄▄▄▄▄▄
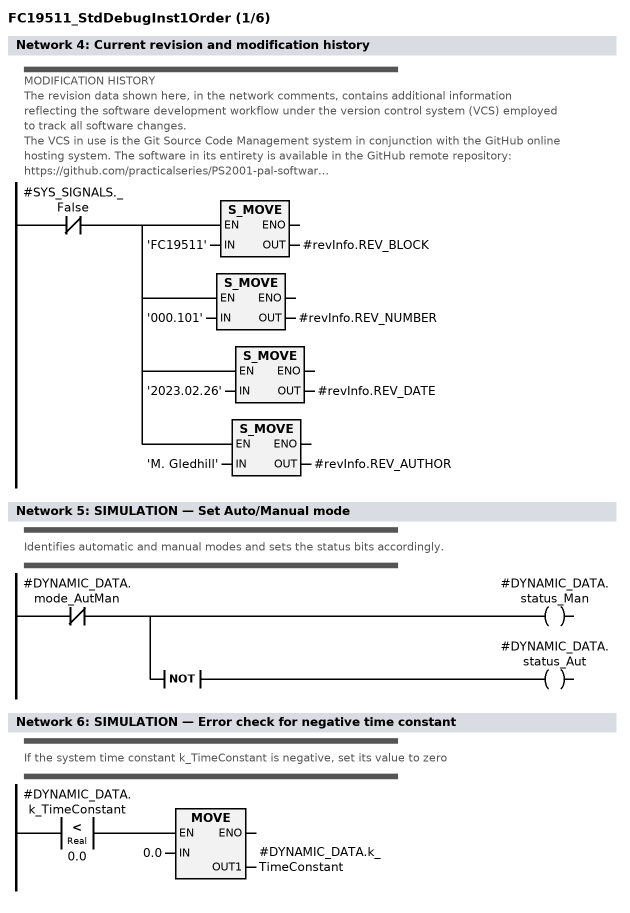
   RUNG wire#powerrail
      I_Contact( #SYS_SIGNALS._False )
      wire#w1
      S_Move(in := 'FC19511', out => #revInfo.REV_BLOCK)
   END_RUNG
   RUNG wire#w1
      S_Move(in := '000.101', out => #revInfo.REV_NUMBER)
   END_RUNG
   RUNG wire#w1
      S_Move(in := '2023.02.26', out => #revInfo.REV_DATE)
   END_RUNG
   RUNG wire#w1
      S_Move(in := 'M. Gledhill', out => #revInfo.REV_AUTHOR)
   END_RUNG
   // the same network as SCL:
   IF NOT #SYS_SIGNALS._False THEN
       #revInfo.REV_BLOCK := 'FC19511';
       #revInfo.REV_NUMBER := '000.101';
       #revInfo.REV_DATE := '2023.02.26';
       #revInfo.REV_AUTHOR := 'M. Gledhill';
   END_IF;
END_REGION

REGION Network 5: SIMULATION — Set Auto/Manual mode
   // ▀▀▀▀▀▀▀▀▀▀▀▀▀▀▀▀▀▀▀▀▀▀▀▀▀▀▀▀▀▀▀▀▀▀▀▀▀▀▀▀▀▀▀▀
   // Identifies automatic and manual modes and sets the status bits accordingly.
   // ▄▄▄▄▄▄▄▄▄▄▄▄▄▄▄▄▄▄▄▄▄▄▄▄▄▄▄▄▄▄▄▄▄▄▄▄▄▄▄▄▄▄▄▄
   RUNG wire#powerrail
      I_Contact( #DYNAMIC_DATA.mode_AutMan )
      wire#w1
      Coil( #DYNAMIC_DATA.status_Man )
   END_RUNG
   RUNG wire#w1
      Not()
      Coil( #DYNAMIC_DATA.status_Aut )
   END_RUNG
   // the same network as SCL:
   #DYNAMIC_DATA.status_Man := NOT #DYNAMIC_DATA.mode_AutMan;
   #DYNAMIC_DATA.status_Aut := NOT (NOT #DYNAMIC_DATA.mode_AutMan);
END_REGION

REGION Network 6: SIMULATION — Error check for negative time constant
   // ▀▀▀▀▀▀▀▀▀▀▀▀▀▀▀▀▀▀▀▀▀▀▀▀▀▀▀▀▀▀▀▀▀▀▀▀▀▀▀▀▀▀▀▀
   // If the system time constant k_TimeConstant is negative, set its value to zero
   // ▄▄▄▄▄▄▄▄▄▄▄▄▄▄▄▄▄▄▄▄▄▄▄▄▄▄▄▄▄▄▄▄▄▄▄▄▄▄▄▄▄▄▄▄
   RUNG wire#powerrail
      { S7_Templates := "SrcType := Real" } LT_Contact(in1 := #DYNAMIC_DATA.k_TimeConstant, in2 := 0.0)
      Move(in := 0.0, out1 => #DYNAMIC_DATA.k_TimeConstant)
   END_RUNG
   // the same network as SCL:
   IF #DYNAMIC_DATA.k_TimeConstant < 0.0 THEN #DYNAMIC_DATA.k_TimeConstant := 0.0; END_IF;
END_REGION

REGION Network 7: SIMULATION INACTIVE — Reset data — Block end
   // ▀▀▀▀▀▀▀▀▀▀▀▀▀▀▀▀▀▀▀▀▀▀▀▀▀▀▀▀▀▀▀▀▀▀▀▀▀▀▀▀▀▀▀▀
   // If the simulation is not running (TRIGGER = 0), set status to stopped and reset all calculated data
   // and status signals.
   // 
   // Set the previous time to the current CPU time (in readiness for the start of the simulation)
   // 
   // Set the OUTPUT, actual_Output and actual_PrevOutput to zero
   // 
   // If the simulation is not running, the block will terminate at this point.
   // ▄▄▄▄▄▄▄▄▄▄▄▄▄▄▄▄▄▄▄▄▄▄▄▄▄▄▄▄▄▄▄▄▄▄▄▄▄▄▄▄▄▄▄▄
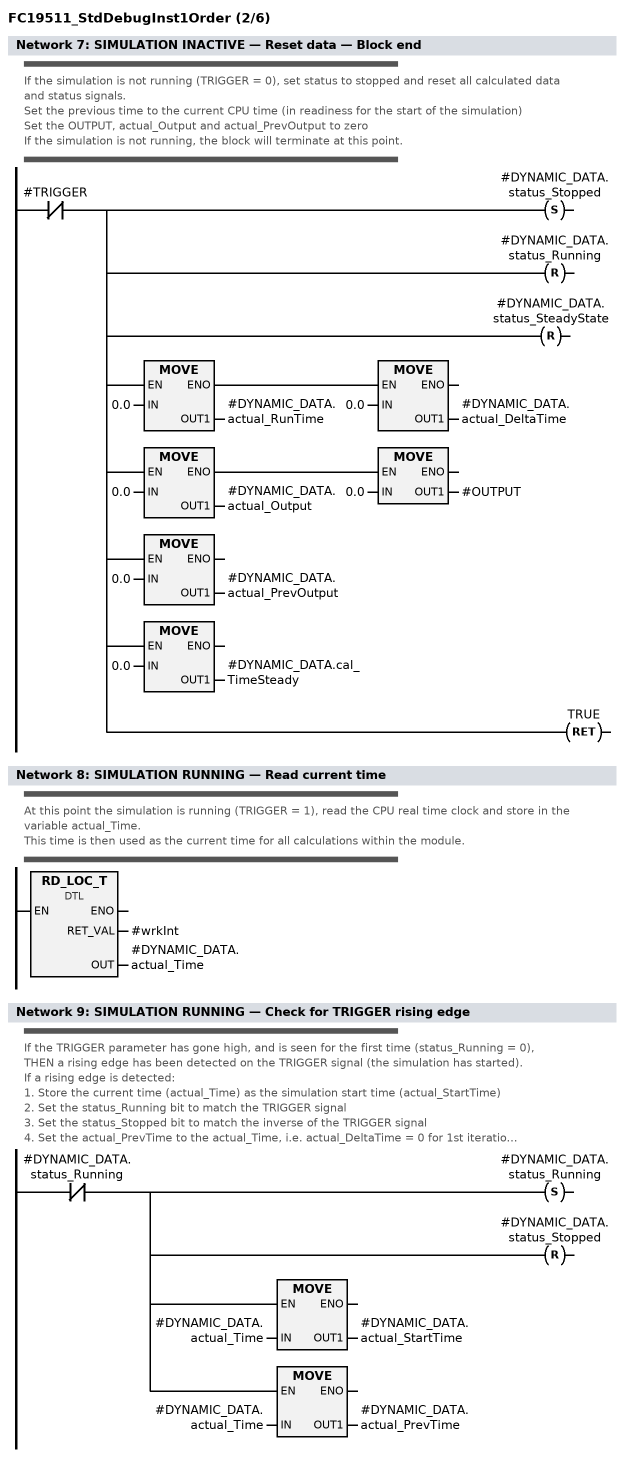
   IF NOT #TRIGGER THEN
       #DYNAMIC_DATA.status_Stopped := TRUE;
       #DYNAMIC_DATA.status_Running := FALSE;
       #DYNAMIC_DATA.status_SteadyState := FALSE;
       #DYNAMIC_DATA.actual_RunTime := 0.0;
       #DYNAMIC_DATA.actual_DeltaTime := 0.0;
       #DYNAMIC_DATA.actual_Output := 0.0;
       #OUTPUT := 0.0;
       #DYNAMIC_DATA.actual_PrevOutput := 0.0;
       #DYNAMIC_DATA.cal_TimeSteady := 0.0;
       ENO := TRUE;
       RETURN;
   END_IF;
END_REGION

REGION Network 8: SIMULATION RUNNING — Read current time
   // ▀▀▀▀▀▀▀▀▀▀▀▀▀▀▀▀▀▀▀▀▀▀▀▀▀▀▀▀▀▀▀▀▀▀▀▀▀▀▀▀▀▀▀▀
   // At this point the simulation is running (TRIGGER = 1), read the CPU real time clock and store in the 
   // variable actual_Time.
   // 
   // This time is then used as the current time for all calculations within the module.
   // ▄▄▄▄▄▄▄▄▄▄▄▄▄▄▄▄▄▄▄▄▄▄▄▄▄▄▄▄▄▄▄▄▄▄▄▄▄▄▄▄▄▄▄▄
   RUNG wire#powerrail
      { S7_Templates := "date_type := DTL" } RD_LOC_T(RET_VAL => #wrkInt, OUT => #DYNAMIC_DATA.actual_Time)
   END_RUNG
   // the same network as SCL:
   #wrkInt := RD_LOC_T(OUT => #DYNAMIC_DATA.actual_Time);
END_REGION

REGION Network 9: SIMULATION RUNNING — Check for TRIGGER rising edge
   // ▀▀▀▀▀▀▀▀▀▀▀▀▀▀▀▀▀▀▀▀▀▀▀▀▀▀▀▀▀▀▀▀▀▀▀▀▀▀▀▀▀▀▀▀
   // If the TRIGGER parameter has gone high, and is seen for the first time (status_Running = 0),
   // THEN a rising edge has been detected on the TRIGGER signal (the simulation has started).
   // 
   // If a rising edge is detected:
   //   1. Store the current time (actual_Time) as the simulation start time (actual_StartTime)
   //   2. Set the status_Running bit to match the TRIGGER signal
   //   3. Set the status_Stopped bit to match the inverse of the TRIGGER signal
   //   4. Set the actual_PrevTime to the actual_Time, i.e. actual_DeltaTime = 0 for 1st iteration
   // ▄▄▄▄▄▄▄▄▄▄▄▄▄▄▄▄▄▄▄▄▄▄▄▄▄▄▄▄▄▄▄▄▄▄▄▄▄▄▄▄▄▄▄▄
   RUNG wire#powerrail
      I_Contact( #DYNAMIC_DATA.status_Running )
      wire#w1
      S_Coil( #DYNAMIC_DATA.status_Running )
   END_RUNG
   RUNG wire#w1
      R_Coil( #DYNAMIC_DATA.status_Stopped )
   END_RUNG
   RUNG wire#w1
      Move(in := #DYNAMIC_DATA.actual_Time, out1 => #DYNAMIC_DATA.actual_StartTime)
   END_RUNG
   RUNG wire#w1
      Move(in := #DYNAMIC_DATA.actual_Time, out1 => #DYNAMIC_DATA.actual_PrevTime)
   END_RUNG
   // the same network as SCL:
   #_w1 := NOT #DYNAMIC_DATA.status_Running;
   IF #_w1 THEN
       #DYNAMIC_DATA.status_Running := TRUE;
       #DYNAMIC_DATA.status_Stopped := FALSE;
       #DYNAMIC_DATA.actual_StartTime := #DYNAMIC_DATA.actual_Time;
       #DYNAMIC_DATA.actual_PrevTime := #DYNAMIC_DATA.actual_Time;
   END_IF;
END_REGION

REGION Network 10: SIMULATION RUNNING — Calculate current elapsed time
   // ▀▀▀▀▀▀▀▀▀▀▀▀▀▀▀▀▀▀▀▀▀▀▀▀▀▀▀▀▀▀▀▀▀▀▀▀▀▀▀▀▀▀▀▀
   // If the TRIGGER parameter is high (the simulation is running), then:
   // Subtract the start time from the current time to give the current elapsed time (wrkElapsedTime)
   // 
   // The elapsed time is calculated in the LTIme format
   // ▄▄▄▄▄▄▄▄▄▄▄▄▄▄▄▄▄▄▄▄▄▄▄▄▄▄▄▄▄▄▄▄▄▄▄▄▄▄▄▄▄▄▄▄
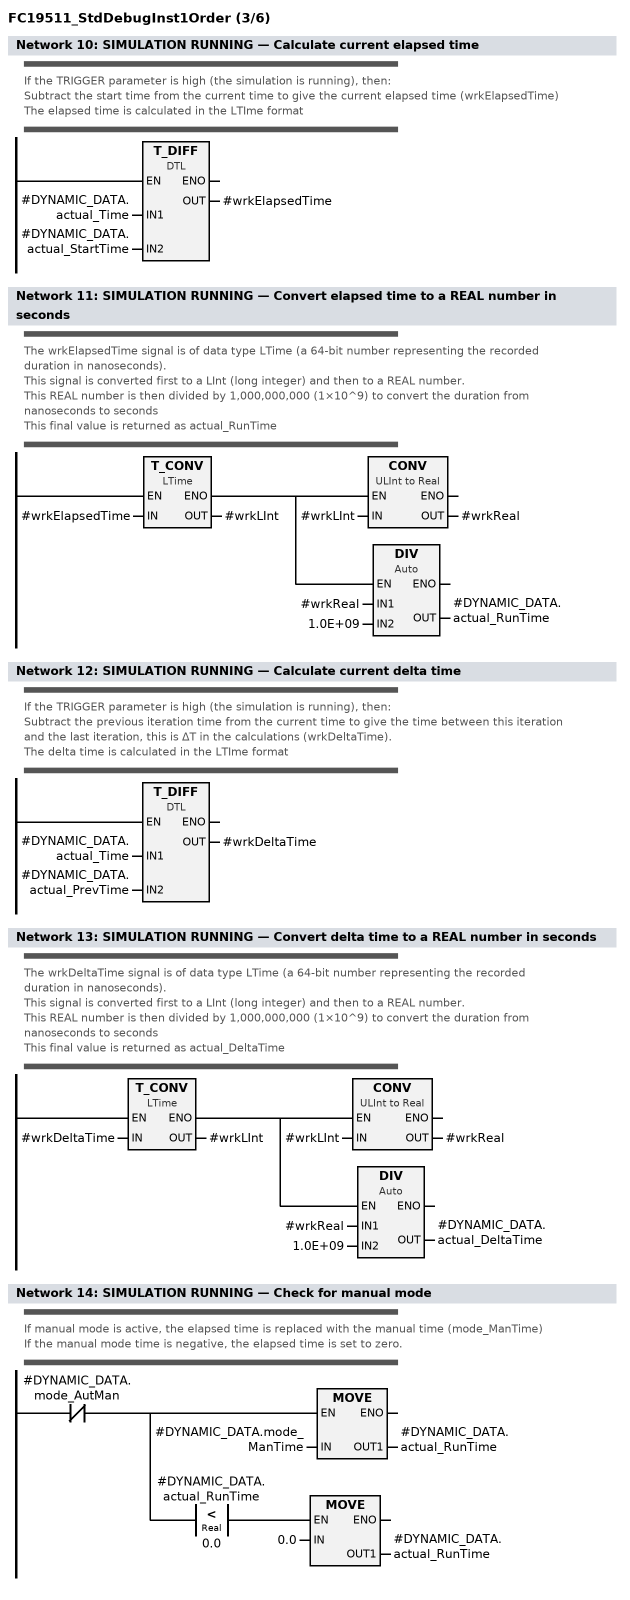
   RUNG wire#powerrail
      { S7_Templates := "[date_type := DTL, time_type := LTime]" } T_DIFF(IN1 := #DYNAMIC_DATA.actual_Time, IN2 := #DYNAMIC_DATA.actual_StartTime, OUT => #wrkElapsedTime)
   END_RUNG
   // the same network as SCL:
   T_DIFF(IN1 := #DYNAMIC_DATA.actual_Time, IN2 := #DYNAMIC_DATA.actual_StartTime, OUT => #wrkElapsedTime);
END_REGION

REGION Network 11: SIMULATION RUNNING — Convert elapsed time to a REAL number in seconds
   // ▀▀▀▀▀▀▀▀▀▀▀▀▀▀▀▀▀▀▀▀▀▀▀▀▀▀▀▀▀▀▀▀▀▀▀▀▀▀▀▀▀▀▀▀
   // The wrkElapsedTime signal is of data type LTime (a 64-bit number representing the recorded
   // duration in nanoseconds).
   // 
   // This signal is converted first to a LInt (long integer) and then to a REAL number.
   // 
   // This REAL number is then divided by 1,000,000,000 (1×10^9) to convert the duration from 
   // nanoseconds to seconds
   // 
   // This final value is returned as actual_RunTime
   // ▄▄▄▄▄▄▄▄▄▄▄▄▄▄▄▄▄▄▄▄▄▄▄▄▄▄▄▄▄▄▄▄▄▄▄▄▄▄▄▄▄▄▄▄
   RUNG wire#powerrail
      { S7_Templates := "[src_type := LTime, dest_type := ULInt]" } T_CONV(IN := #wrkElapsedTime, OUT => #wrkLInt)
      wire#w1
      { S7_Templates := "[SrcType := ULInt, DestType := Real]" } Convert(in := #wrkLInt, out => #wrkReal)
   END_RUNG
   RUNG wire#w1
      Div(in1 := #wrkReal, in2 := 1.0E+09, out => #DYNAMIC_DATA.actual_RunTime)
   END_RUNG
   // the same network as SCL:
   T_CONV(IN := #wrkElapsedTime, OUT => #wrkLInt, ENO => #_w1);
   IF #_w1 THEN
       #wrkReal := ULINT_TO_REAL(#wrkLInt);
       #DYNAMIC_DATA.actual_RunTime := #wrkReal / 1.0E+09;
   END_IF;
END_REGION

REGION Network 12: SIMULATION RUNNING — Calculate current delta time
   // ▀▀▀▀▀▀▀▀▀▀▀▀▀▀▀▀▀▀▀▀▀▀▀▀▀▀▀▀▀▀▀▀▀▀▀▀▀▀▀▀▀▀▀▀
   // If the TRIGGER parameter is high (the simulation is running), then:
   // Subtract the previous iteration time from the current time to give the time between this iteration
   // and the last iteration, this is ΔT in the calculations (wrkDeltaTime).
   // 
   // The delta time is calculated in the LTIme format
   // ▄▄▄▄▄▄▄▄▄▄▄▄▄▄▄▄▄▄▄▄▄▄▄▄▄▄▄▄▄▄▄▄▄▄▄▄▄▄▄▄▄▄▄▄
   RUNG wire#powerrail
      { S7_Templates := "[date_type := DTL, time_type := LTime]" } T_DIFF(IN1 := #DYNAMIC_DATA.actual_Time, IN2 := #DYNAMIC_DATA.actual_PrevTime, OUT => #wrkDeltaTime)
   END_RUNG
   // the same network as SCL:
   T_DIFF(IN1 := #DYNAMIC_DATA.actual_Time, IN2 := #DYNAMIC_DATA.actual_PrevTime, OUT => #wrkDeltaTime);
END_REGION

REGION Network 13: SIMULATION RUNNING — Convert delta time to a REAL number in seconds
   // ▀▀▀▀▀▀▀▀▀▀▀▀▀▀▀▀▀▀▀▀▀▀▀▀▀▀▀▀▀▀▀▀▀▀▀▀▀▀▀▀▀▀▀▀
   // The wrkDeltaTime signal is of data type LTime (a 64-bit number representing the recorded
   // duration in nanoseconds).
   // 
   // This signal is converted first to a LInt (long integer) and then to a REAL number.
   // 
   // This REAL number is then divided by 1,000,000,000 (1×10^9) to convert the duration from 
   // nanoseconds to seconds
   // 
   // This final value is returned as actual_DeltaTime
   // ▄▄▄▄▄▄▄▄▄▄▄▄▄▄▄▄▄▄▄▄▄▄▄▄▄▄▄▄▄▄▄▄▄▄▄▄▄▄▄▄▄▄▄▄
   RUNG wire#powerrail
      { S7_Templates := "[src_type := LTime, dest_type := ULInt]" } T_CONV(IN := #wrkDeltaTime, OUT => #wrkLInt)
      wire#w1
      { S7_Templates := "[SrcType := ULInt, DestType := Real]" } Convert(in := #wrkLInt, out => #wrkReal)
   END_RUNG
   RUNG wire#w1
      Div(in1 := #wrkReal, in2 := 1.0E+09, out => #DYNAMIC_DATA.actual_DeltaTime)
   END_RUNG
   // the same network as SCL:
   T_CONV(IN := #wrkDeltaTime, OUT => #wrkLInt, ENO => #_w1);
   IF #_w1 THEN
       #wrkReal := ULINT_TO_REAL(#wrkLInt);
       #DYNAMIC_DATA.actual_DeltaTime := #wrkReal / 1.0E+09;
   END_IF;
END_REGION

REGION Network 14: SIMULATION RUNNING — Check for manual mode
   // ▀▀▀▀▀▀▀▀▀▀▀▀▀▀▀▀▀▀▀▀▀▀▀▀▀▀▀▀▀▀▀▀▀▀▀▀▀▀▀▀▀▀▀▀
   // If manual mode is active, the elapsed time is replaced with the manual time (mode_ManTime)
   // 
   // If the manual mode time is negative, the elapsed time is set to zero.
   // ▄▄▄▄▄▄▄▄▄▄▄▄▄▄▄▄▄▄▄▄▄▄▄▄▄▄▄▄▄▄▄▄▄▄▄▄▄▄▄▄▄▄▄▄
   RUNG wire#powerrail
      I_Contact( #DYNAMIC_DATA.mode_AutMan )
      wire#w1
      Move(in := #DYNAMIC_DATA.mode_ManTime, out1 => #DYNAMIC_DATA.actual_RunTime)
   END_RUNG
   RUNG wire#w1
      { S7_Templates := "SrcType := Real" } LT_Contact(in1 := #DYNAMIC_DATA.actual_RunTime, in2 := 0.0)
      Move(in := 0.0, out1 => #DYNAMIC_DATA.actual_RunTime)
   END_RUNG
   // the same network as SCL:
   #_w1 := NOT #DYNAMIC_DATA.mode_AutMan;
   IF #_w1 THEN #DYNAMIC_DATA.actual_RunTime := #DYNAMIC_DATA.mode_ManTime; END_IF;
   IF #_w1 AND (#DYNAMIC_DATA.actual_RunTime < 0.0) THEN #DYNAMIC_DATA.actual_RunTime := 0.0; END_IF;
END_REGION

REGION Network 15: SIMULATION RUNNING — Real-time simulation calculation
   // ▀▀▀▀▀▀▀▀▀▀▀▀▀▀▀▀▀▀▀▀▀▀▀▀▀▀▀▀▀▀▀▀▀▀▀▀▀▀▀▀▀▀▀▀
   // If the simulation is running and is in automatic mode, the following iterative, Real-time 
   // simulation calculation is carried out:
   // 
   // CALCULATION:
   //                               ΔT
   //    y[n] = Ka x[n]  ┼ (1-a) y[n-1]   where: a = ----------
   //                             τ+ΔT
   // 
   // Is rendered into the correct format as follows:
   // 
   // 
   //  cal_01 = ΔT             =  actual_DeltaTime
   // 
   //  cal_02 = τ + ΔT             = k_TimeConstant + cal_01
   // 
   //                ΔT
   //  cal_03 = a = ----------          = cal_01 ÷ cal_02
   //                 τ+ΔT
   // 
   //  cal_04 = 1 - a             = 1 - cal_03
   // 
   // 
   //  cal_05 = Kax[n]            = k_Gain × cal_03 × INPUT
   // 
   //  cal_06 = (1-a) y[n-1]          = cal_04 × actual_PrevOutput
   // 
   // 
   //  OUTPUT  = Ka x[n]  ┼ (1-a) y[n-1]      = cal_05 × cal_06
   // 
   // 
   // ▄▄▄▄▄▄▄▄▄▄▄▄▄▄▄▄▄▄▄▄▄▄▄▄▄▄▄▄▄▄▄▄▄▄▄▄▄▄▄▄▄▄▄▄
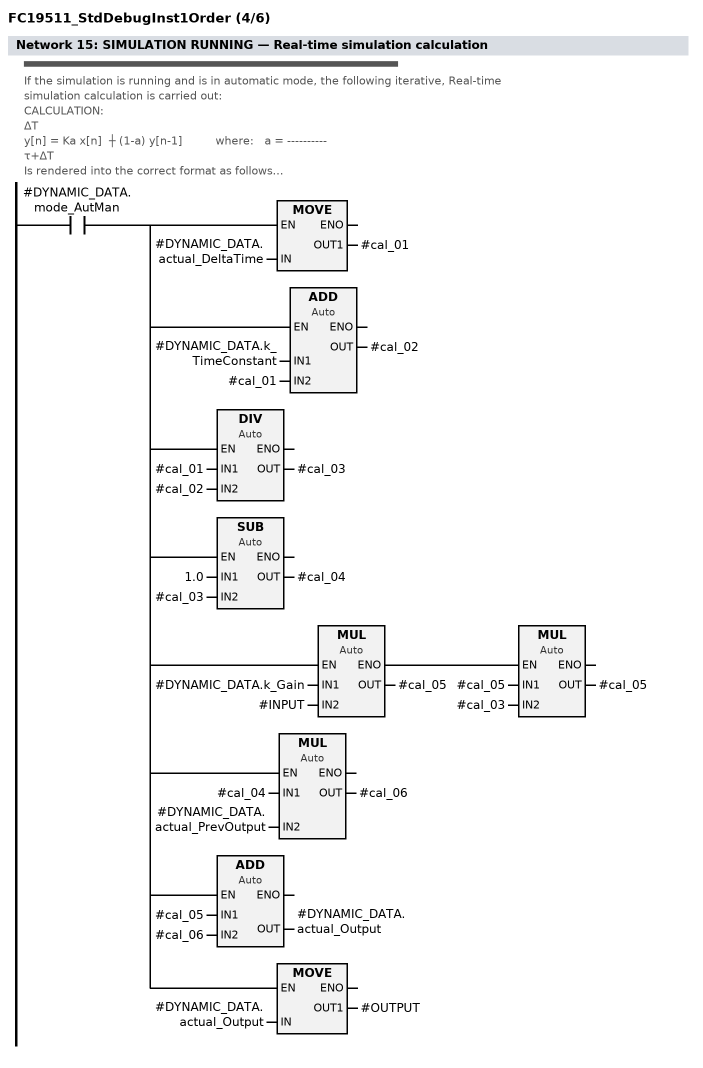
   RUNG wire#powerrail
      Contact( #DYNAMIC_DATA.mode_AutMan )
      wire#w1
      Move(in := #DYNAMIC_DATA.actual_DeltaTime, out1 => #cal_01)
   END_RUNG
   RUNG wire#w1
      Add(in1 := #DYNAMIC_DATA.k_TimeConstant, in2 := #cal_01, out => #cal_02)
   END_RUNG
   RUNG wire#w1
      Div(in1 := #cal_01, in2 := #cal_02, out => #cal_03)
   END_RUNG
   RUNG wire#w1
      Sub(in1 := 1.0, in2 := #cal_03, out => #cal_04)
   END_RUNG
   RUNG wire#w1
      Mul(in1 := #DYNAMIC_DATA.k_Gain, in2 := #INPUT, out => #cal_05)
      Mul(in1 := #cal_05, in2 := #cal_03, out => #cal_05)
   END_RUNG
   RUNG wire#w1
      Mul(in1 := #cal_04, in2 := #DYNAMIC_DATA.actual_PrevOutput, out => #cal_06)
   END_RUNG
   RUNG wire#w1
      Add(in1 := #cal_05, in2 := #cal_06, out => #DYNAMIC_DATA.actual_Output)
   END_RUNG
   RUNG wire#w1
      Move(in := #DYNAMIC_DATA.actual_Output, out1 => #OUTPUT)
   END_RUNG
   // the same network as SCL:
   IF #DYNAMIC_DATA.mode_AutMan THEN
       #cal_01 := #DYNAMIC_DATA.actual_DeltaTime;
       #cal_02 := #DYNAMIC_DATA.k_TimeConstant + #cal_01;
       #cal_03 := #cal_01 / #cal_02;
       #cal_04 := 1.0 - #cal_03;
       #cal_05 := #DYNAMIC_DATA.k_Gain * #INPUT;
       #cal_05 := #cal_05 * #cal_03;
       #cal_06 := #cal_04 * #DYNAMIC_DATA.actual_PrevOutput;
       #DYNAMIC_DATA.actual_Output := #cal_05 + #cal_06;
       #OUTPUT := #DYNAMIC_DATA.actual_Output;
   END_IF;
END_REGION

REGION Network 16: SIMULATION RUNNING — Over damped — Ancillary calculations
   // ▀▀▀▀▀▀▀▀▀▀▀▀▀▀▀▀▀▀▀▀▀▀▀▀▀▀▀▀▀▀▀▀▀▀▀▀▀▀▀▀▀▀▀▀
   // If the simulation is running and is in manual mode, the following discrete manual response to a 
   // step input calculation is carried out:
   // 
   // 
   // CALCULATION:
   // 
   //          ┌      -t/τ  ┐
   //    y(t) = KX│ 1 ─  e   │
   //          └       ┘
   // 
   // 
   // Is rendered into the correct format as follows:
   // 
   // 
   //  cal_01 =  -t/τ            = - 1 × actual_RunTime ÷  k_TimeConstant
   // 
   //          - t/τ
   //  cal_02 = ｅ              = EXP (cal_01)
   // 
   //                - t/τ
   //  cal_03 = 1 ─  ｅ              = 1 - cal_02
   // 
   // 
   //              ┌      -t/τ  ┐
   //  OUTPUT  = KX│ 1 ─  e   │       = k_Gain × INPUT × cal_03
   //              └       ┘
   // 
   // Note:    If k_TimeConstant = 0, cal_01 is set to the value k_NEG_MAX (the largest
   //      negative value available to a real number), preventing divide by zero errors.
   // 
   // ▄▄▄▄▄▄▄▄▄▄▄▄▄▄▄▄▄▄▄▄▄▄▄▄▄▄▄▄▄▄▄▄▄▄▄▄▄▄▄▄▄▄▄▄
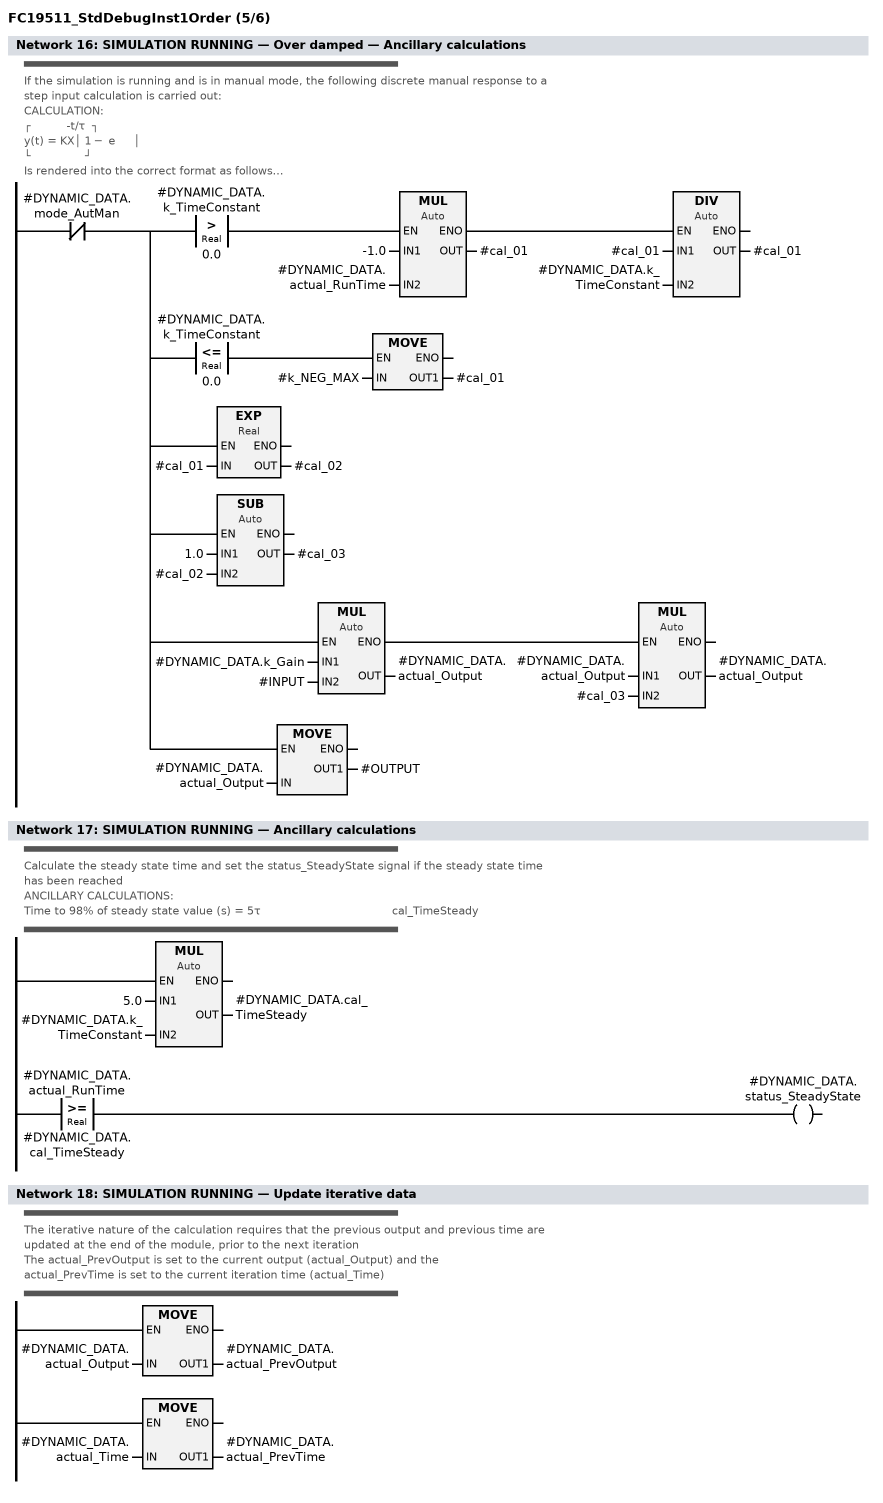
   #_w1 := NOT #DYNAMIC_DATA.mode_AutMan;
   IF #_w1 AND (#DYNAMIC_DATA.k_TimeConstant > 0.0) THEN
       #cal_01 := (-1.0) * #DYNAMIC_DATA.actual_RunTime;
       #cal_01 := #cal_01 / #DYNAMIC_DATA.k_TimeConstant;
   END_IF;
   IF #_w1 AND (#DYNAMIC_DATA.k_TimeConstant <= 0.0) THEN #cal_01 := #k_NEG_MAX; END_IF;
   IF #_w1 THEN
       #cal_02 := EXP(#cal_01);
       #cal_03 := 1.0 - #cal_02;
       #DYNAMIC_DATA.actual_Output := #DYNAMIC_DATA.k_Gain * #INPUT;
       #DYNAMIC_DATA.actual_Output := #DYNAMIC_DATA.actual_Output * #cal_03;
       #OUTPUT := #DYNAMIC_DATA.actual_Output;
   END_IF;
END_REGION

REGION Network 17: SIMULATION RUNNING — Ancillary calculations
   // ▀▀▀▀▀▀▀▀▀▀▀▀▀▀▀▀▀▀▀▀▀▀▀▀▀▀▀▀▀▀▀▀▀▀▀▀▀▀▀▀▀▀▀▀
   // Calculate the steady state time and set the status_SteadyState signal if the steady state time
   // has been reached
   // 
   // 
   // 
   // ANCILLARY CALCULATIONS:
   // 
   //  Time to 98% of steady state value (s) = 5τ              cal_TimeSteady
   // ▄▄▄▄▄▄▄▄▄▄▄▄▄▄▄▄▄▄▄▄▄▄▄▄▄▄▄▄▄▄▄▄▄▄▄▄▄▄▄▄▄▄▄▄
   RUNG wire#powerrail
      Mul(in1 := 5.0, in2 := #DYNAMIC_DATA.k_TimeConstant, out => #DYNAMIC_DATA.cal_TimeSteady)
   END_RUNG
   RUNG wire#powerrail
      { S7_Templates := "SrcType := Real" } GE_Contact(in1 := #DYNAMIC_DATA.actual_RunTime, in2 := #DYNAMIC_DATA.cal_TimeSteady)
      Coil( #DYNAMIC_DATA.status_SteadyState )
   END_RUNG
   // the same network as SCL:
   #DYNAMIC_DATA.cal_TimeSteady := 5.0 * #DYNAMIC_DATA.k_TimeConstant;
   #DYNAMIC_DATA.status_SteadyState := #DYNAMIC_DATA.actual_RunTime >= #DYNAMIC_DATA.cal_TimeSteady;
END_REGION

REGION Network 18: SIMULATION RUNNING — Update iterative data
   // ▀▀▀▀▀▀▀▀▀▀▀▀▀▀▀▀▀▀▀▀▀▀▀▀▀▀▀▀▀▀▀▀▀▀▀▀▀▀▀▀▀▀▀▀
   // The iterative nature of the calculation requires that the previous output and previous time are
   // updated at the end of the module, prior to the next iteration
   // 
   // The actual_PrevOutput is set to the current output (actual_Output) and the
   // actual_PrevTime is set to the current iteration time (actual_Time)
   // ▄▄▄▄▄▄▄▄▄▄▄▄▄▄▄▄▄▄▄▄▄▄▄▄▄▄▄▄▄▄▄▄▄▄▄▄▄▄▄▄▄▄▄▄
   RUNG wire#powerrail
      Move(in := #DYNAMIC_DATA.actual_Output, out1 => #DYNAMIC_DATA.actual_PrevOutput)
   END_RUNG
   RUNG wire#powerrail
      Move(in := #DYNAMIC_DATA.actual_Time, out1 => #DYNAMIC_DATA.actual_PrevTime)
   END_RUNG
   // the same network as SCL:
   #DYNAMIC_DATA.actual_PrevOutput := #DYNAMIC_DATA.actual_Output;
   #DYNAMIC_DATA.actual_PrevTime := #DYNAMIC_DATA.actual_Time;
END_REGION

REGION Network 19: LICENCE AND CONTACT INFORMATION
   // ▀▀▀▀▀▀▀▀▀▀▀▀▀▀▀▀▀▀▀▀▀▀▀▀▀▀▀▀▀▀▀▀▀▀▀▀▀▀▀▀▀▀▀▀
   // LICENCE AND CONTACT INFORMATION
   // 
   // This software and its associated documentation is made available under the MIT Licence:
   // 
   // ════════════════════════════════════════════
   // 
   // The MIT License (MIT)
   // 
   // Copyright © 2020 Michael Gledhill
   // 
   // Permission is hereby granted, free of charge, to any person obtaining a copy of this software 
   // and associated documentation files (the “Software”), to deal in the Software without restriction, 
   // including without limitation the rights to use, copy, modify, merge, publish, distribute, 
   // sublicense, and/or sell copies of the Software, and to permit persons to whom the Software is 
   // furnished to do so, subject to the following conditions: 
   // 
   // The above copyright notice and this permission notice shall be included in all copies or 
   // substantial portions of the Software.
   // 
   // THE SOFTWARE IS PROVIDED “AS IS”, WITHOUT WARRANTY OF ANY KIND, EXPRESS OR IMPLIED, 
   // INCLUDING BUT NOT LIMITED TO THE WARRANTIES OF MERCHANTABILITY, FITNESS FOR A 
   // PARTICULAR PURPOSE AND NON-INFRINGEMENT. IN NO EVENT SHALL THE AUTHORS OR COPYRIGHT 
   // HOLDERS BE LIABLE FOR ANY CLAIM, DAMAGES OR OTHER LIABILITY, WHETHER IN AN ACTION OF 
   // CONTRACT, TORT OR OTHERWISE, ARISING FROM, OUT OF OR IN CONNECTION WITH THE SOFTWARE 
   // OR THE USE OR OTHER DEALINGS IN THE SOFTWARE.
   // 
   // ════════════════════════════════════════════
   //                    ┌────────────┐
   // You can reach the author by email here:   │  mg@practicalseries.com  │
   //                    └────────────┘
   // Questions, corrections, constructive criticism and complaints (polite ones) are invited.
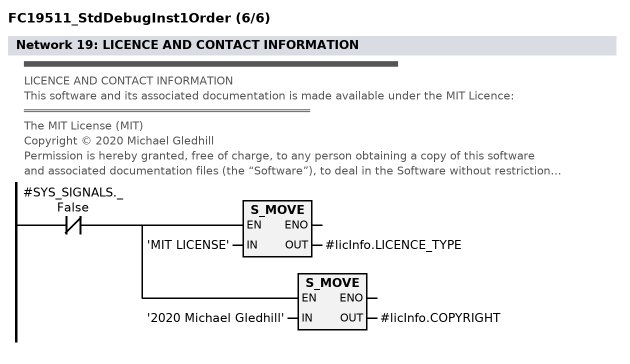
   RUNG wire#powerrail
      I_Contact( #SYS_SIGNALS._False )
      wire#w1
      S_Move(in := 'MIT LICENSE', out => #licInfo.LICENCE_TYPE)
   END_RUNG
   RUNG wire#w1
      S_Move(in := '2020 Michael Gledhill', out => #licInfo.COPYRIGHT)
   END_RUNG
   // the same network as SCL:
   IF NOT #SYS_SIGNALS._False THEN
       #licInfo.LICENCE_TYPE := 'MIT LICENSE';
       #licInfo.COPYRIGHT := '2020 Michael Gledhill';
   END_IF;
END_REGION
END_FUNCTION
